# B&R Automation Studio project CControl_Gschneitner (part 8)

#### fbRestzeit.st
```iecst
(* Funktionsbaustein zur Berechnung der Restzeit Lauf/Pause aus 24h Zeitfenstern (BOOL [24]) *)
FUNCTION_BLOCK fbRestzeit

	IF Freigabe THEN

		//Variable setzen, wenn Zeitfenster aktiv
		ZeitfensterAktiv	:= ZeitfensterIn[AktuelleStunde];

		//Zeitfenster ist aktiv -> Restzeit Lauf berechnen *********************************************************
		IF ZeitfensterAktiv THEN

			//Änderung von Struktur Zeitfenster erkennen
			loc_Aenderung := memcmp(ADR(ZeitfensterIn), ADR(MEM_ZeitfensterIn), SIZEOF(ZeitfensterIn));
			IF loc_Aenderung <> 0 OR loc_firstInitLauf THEN
				loc_firstInitLauf := FALSE;
				loc_StundeEndeZeitfTag := 23;
				loc_StundeEndeZeitfFolgetag := 23;
				memcpy(ADR(MEM_ZeitfensterIn), ADR(ZeitfensterIn), SIZEOF(MEM_ZeitfensterIn));
			END_IF

			//Minuten Rest aktueller Tag berechnen
			loc_MinutenRestTag	:= 60 - AktuelleMinute;
			FOR i:= AktuelleStunde + 1 TO loc_StundeEndeZeitfTag DO
				IF ZeitfensterIn[i] = TRUE THEN
					loc_MinutenRestTag	:= loc_MinutenRestTag + 60;
				ELSE
					loc_StundeEndeZeitfTag := i;
				END_IF
			END_FOR

			//Minuten Rest Folgetag berechnen, wenn aktuelles Zeitfenster bis zum Ende des Tages aktiv ist
			loc_MinutenRestFolgetag := 0;
			IF loc_StundeEndeZeitfTag = 23 THEN
				FOR ii:= 0 TO loc_StundeEndeZeitfFolgetag DO
					IF ZeitfensterIn[ii] = TRUE THEN
						loc_MinutenRestFolgetag	:= loc_MinutenRestFolgetag + 60;
					ELSE
						loc_StundeEndeZeitfFolgetag := ii;
					END_IF
				END_FOR
			ELSE
				loc_MinutenRestFolgetag := 0;
				loc_StundeEndeZeitfFolgetag := 23;
			END_IF

			//Gesamtzeit Minuten Tag + Folgetag
			loc_MinutenRestGesamt := loc_MinutenRestTag + loc_MinutenRestFolgetag;

			//Ausgabe Restzeit in Stunden und Minuten
			loc_RestzeitStunden		:= loc_MinutenRestGesamt / 60;
			//Wenn Restzeit Stunden > 24h, Ausgabe Stunden = 255 (keine Anzeige in Visu)
			IF loc_RestzeitStunden <= 24 THEN
				RestzeitStundenOut		:= ABS(loc_RestzeitStunden);
				RestzeitMinutenOut		:= loc_MinutenRestGesamt - (RestzeitStundenOut * 60);
			ELSE
				RestzeitStundenOut		:= 65535;
				RestzeitMinutenOut		:= 65535;
			END_IF

			loc_firstInitPause := TRUE;

		//Zeitfenster nicht aktiv -> Restzeit Pause berechnen *********************************************************
		ELSE

			//Änderung von Struktur Zeitfenster erkennen
			loc_Aenderung := memcmp(ADR(ZeitfensterIn), ADR(MEM_ZeitfensterIn), SIZEOF(ZeitfensterIn));
			IF loc_Aenderung <> 0 OR loc_firstInitPause THEN
				loc_firstInitPause := FALSE;
				loc_StundeEndeZeitfTag := 23;
				loc_StundeEndeZeitfFolgetag := 23;
				memcpy(ADR(MEM_ZeitfensterIn), ADR(ZeitfensterIn), SIZEOF(MEM_ZeitfensterIn));
			END_IF

			//Minuten Rest aktueller Tag berechnen
			loc_MinutenRestTag	:= 60 - AktuelleMinute;
			FOR i:= AktuelleStunde + 1 TO loc_StundeEndeZeitfTag DO
				IF ZeitfensterIn[i] = FALSE THEN
					loc_MinutenRestTag	:= loc_MinutenRestTag + 60;
				ELSE
					loc_StundeEndeZeitfTag := i;
				END_IF
			END_FOR

			//Minuten Rest Folgetag berechnen, wenn aktuelles Zeitfenster bis zum Ende des Tages inaktiv ist
			loc_MinutenRestFolgetag := 0;
			IF loc_StundeEndeZeitfTag = 23 THEN
				FOR ii:= 0 TO loc_StundeEndeZeitfFolgetag DO
					IF ZeitfensterIn[ii] = FALSE THEN
						loc_MinutenRestFolgetag	:= loc_MinutenRestFolgetag + 60;
					ELSE
						loc_StundeEndeZeitfFolgetag := ii;
					END_IF
				END_FOR
			ELSE
				loc_MinutenRestFolgetag := 0;
				loc_StundeEndeZeitfFolgetag := 23;
			END_IF

			//Gesamtzeit Minuten Tag + Folgetag
			loc_MinutenRestGesamt := loc_MinutenRestTag + loc_MinutenRestFolgetag;

			//Ausgabe Restzeit in Stunden und Minuten
			loc_RestzeitStunden		:= loc_MinutenRestGesamt / 60;

			//Wenn Restzeit Stunden > 24h, Ausgabe Stunden = 65535 (keine Anzeige in Visu)
			IF loc_RestzeitStunden <= 24 THEN
				RestzeitStundenOut		:= ABS(loc_RestzeitStunden);
				RestzeitMinutenOut		:= loc_MinutenRestGesamt - (RestzeitStundenOut * 60);
			ELSE
				RestzeitStundenOut		:= 65535;
				RestzeitMinutenOut		:= 65535;
			END_IF

			loc_firstInitLauf := TRUE;

		END_IF

	//Keine Freigabe Baustein
	ELSE

		loc_firstInitLauf	:= TRUE;
		loc_firstInitPause	:= TRUE;
		RestzeitMinutenOut	:= 65535;
		RestzeitStundenOut	:= 65535;

	END_IF

END_FUNCTION_BLOCK
```

### Library Logical/Libraries/IecCheck (IEC)
Depends on: sys_lib, AsBrStr

#### IecCheck.fun - Exported functions and function blocks
```iecst
FUNCTION CheckDivSint : SINT (* Check divisor for SINT division *)
	VAR_INPUT
		divisor : SINT;
	END_VAR
END_FUNCTION

FUNCTION CheckDivUsint : USINT (* Check divisor for USINT division *)
	VAR_INPUT
		divisor : USINT;
	END_VAR
END_FUNCTION

FUNCTION CheckDivInt : INT (* Check divisor for INT division *)
	VAR_INPUT
		divisor : INT;
	END_VAR
END_FUNCTION

FUNCTION CheckDivUint : UINT (* Check divisor for UINT division *)
	VAR_INPUT
		divisor : UINT;
	END_VAR
END_FUNCTION

FUNCTION CheckDivDint : DINT (* Check divisor for DINT division *)
	VAR_INPUT
		divisor : DINT;
	END_VAR
END_FUNCTION

FUNCTION CheckDivUdint : UDINT (* Check divisor for UDINT division *)
	VAR_INPUT
		divisor : UDINT;
	END_VAR
END_FUNCTION

FUNCTION CheckDivReal : REAL (* Check divisor for REAL division *)
	VAR_INPUT
		divisor : REAL;
	END_VAR
END_FUNCTION

FUNCTION CheckDivLReal : LREAL (* Check divisor for LREAL division, not available for SG3 and SGC *)
	VAR_INPUT
		divisor : LREAL;
	END_VAR
END_FUNCTION

FUNCTION CheckBounds : DINT (* Check range for array access *)
	VAR_INPUT
		index : DINT;
		lower : DINT;
		upper : DINT;
	END_VAR
END_FUNCTION

FUNCTION CheckRange : DINT (* Check range for enumeration *)
	VAR_INPUT
		value : DINT;
		lower : DINT;
		upper : DINT;
	END_VAR
END_FUNCTION

FUNCTION CheckSignedSubrange : DINT (* Check range for subrange of signed data types *)
	VAR_INPUT
		value : DINT;
		lower : DINT;
		upper : DINT;
	END_VAR
END_FUNCTION

FUNCTION CheckUnsignedSubrange : UDINT (* Check range for subrange of unsigned data types *)
	VAR_INPUT
		value : UDINT;
		lower : UDINT;
		upper : UDINT;
	END_VAR
END_FUNCTION

FUNCTION CheckReadAccess : UDINT (* Check address when reading dynamic variables *)
	VAR_INPUT
		address : UDINT;
	END_VAR
END_FUNCTION

FUNCTION CheckWriteAccess : UDINT (* Check address when writing dynamic variables *)
	VAR_INPUT
		address : UDINT;
	END_VAR
END_FUNCTION

FUNCTION MakeEntry : UDINT (* Makes an entry (log book entry) in the error log book *)
	VAR
		taskname : STRING[30];
		group : USINT;
		status_name : UINT;
		out_text : STRING[80];
	END_VAR
	VAR_INPUT
		number : UINT;
		index : DINT;
		text : STRING[50];
	END_VAR
END_FUNCTION
```

#### IecCheck.st - Implementation file
```iecst
(* Check divisor for SINT division *)
FUNCTION CheckDivSint
	IF divisor=0 THEN
		CheckDivSint:=1;
		MakeEntry(55555,divisor,'CheckDivSint');
	ELSE
		CheckDivSint:=divisor;
	END_IF
END_FUNCTION

(* Check divisor for USINT division *)
FUNCTION CheckDivUsint
	IF divisor=0 THEN
		CheckDivUsint:=1;
		MakeEntry(55555,divisor,'CheckDivUsint');
	ELSE
		CheckDivUsint:=divisor;
	END_IF
END_FUNCTION

(* Check divisor for INT division *)
FUNCTION CheckDivInt
	IF divisor=0 THEN
		CheckDivInt:=1;
		MakeEntry(55555,divisor,'CheckDivInt');
	ELSE
		CheckDivInt:=divisor;
	END_IF
END_FUNCTION

(* Check divisor for UINT division *)
FUNCTION CheckDivUint
	IF divisor=0 THEN
		CheckDivUint:=1;
		MakeEntry(55555,divisor,'CheckDivUint');
	ELSE
		CheckDivUint:=divisor;
	END_IF
END_FUNCTION

(* Check divisor for DINT division *)
FUNCTION CheckDivDint
	IF divisor=0 THEN
		CheckDivDint:=1;
		MakeEntry(55555,divisor,'CheckDivDint');
	ELSE
		CheckDivDint:=divisor;
	END_IF
END_FUNCTION

(* Check divisor for UDINT division *)
FUNCTION CheckDivUdint
	IF divisor=0 THEN
		CheckDivUdint:=1;
		MakeEntry(55555,divisor,'CheckDivUdint');
	ELSE
		CheckDivUdint:=divisor;
	END_IF
END_FUNCTION

(* Check divisor for REAL division *)
FUNCTION CheckDivReal
	IF divisor=0 THEN
		CheckDivReal:=1;
		MakeEntry(55555,0,'CheckDivReal');
	ELSE
		CheckDivReal:=divisor;
	END_IF
END_FUNCTION

(* Check divisor for LREAL division *)
FUNCTION CheckDivLReal
	IF divisor=0 THEN
		CheckDivLReal:=1;
		MakeEntry(55555,0,'CheckDivLReal');
	ELSE
		CheckDivLReal:=divisor;
	END_IF
END_FUNCTION

(* Check range for array access *)
FUNCTION CheckBounds
	IF index < lower THEN
		CheckBounds := lower;
		MakeEntry(55555,index,'CheckBounds');
	ELSIF index > upper THEN
		CheckBounds := upper;
		MakeEntry(55555,index,'CheckBounds');
	ELSE
		CheckBounds := index;
	END_IF
END_FUNCTION

(* Check range for enumeration *)
FUNCTION CheckRange
	IF value < lower THEN
		CheckRange := lower;
		MakeEntry(55555,value,'CheckRange');
	ELSIF value > upper THEN
		CheckRange := upper;
		MakeEntry(55555,value,'CheckRange');
	ELSE
		CheckRange := value;
	END_IF
END_FUNCTION

(* Check range for subrange of signed data types *)
FUNCTION CheckSignedSubrange
	IF value < lower THEN
		CheckSignedSubrange := lower;
		MakeEntry(55555,value,'CheckSignedSubrange');
	ELSIF value > upper THEN
		CheckSignedSubrange := upper;
		MakeEntry(55555,value,'CheckSignedSubrange');
	ELSE
		CheckSignedSubrange := value;
	END_IF
END_FUNCTION

(* Check range for subrange of unsigned data types *)
FUNCTION CheckUnsignedSubrange
	IF value < lower THEN
		CheckUnsignedSubrange := lower;
		MakeEntry(55555,value,'CheckUnsignedSubrange');
	ELSIF value > upper THEN
		CheckUnsignedSubrange := upper;
		MakeEntry(55555,value,'CheckUnsignedSubrange');
	ELSE
		CheckUnsignedSubrange := value;
	END_IF
END_FUNCTION

(* Check address when reading dynamic variables *)
FUNCTION CheckReadAccess
	IF address=0 THEN
		(* TODO: Insert an appropriate code, see AutomationStudio help for further information *)
		MakeEntry(55555,address,'Read from NULL');
	END_IF

	CheckReadAccess:=0;
END_FUNCTION

(* Check address when writing dynamic variables *)
FUNCTION CheckWriteAccess
	IF address=0 THEN
		(* TODO: Insert an appropriate code, see AutomationStudio help for further information *)
		MakeEntry(55555,address,'Write to NULL');
	END_IF

	CheckWriteAccess:=0;
END_FUNCTION

(* Makes an entry (log book entry) in the error log book *)
FUNCTION MakeEntry
		status_name := ST_name(0,ADR(taskname),ADR(group));

		brsstrcpy(ADR(out_text),ADR(text));
		brsstrcat(ADR(out_text),ADR(' > in task > '));
  		brsstrcat(ADR(out_text),ADR(taskname));
		MakeEntry := ADR(out_text);
		ERRxfatal(number,index,ADR(out_text));
END_FUNCTION
```

### Library Logical/Libraries/CControl (IEC)

#### CControl.fun - Exported functions and function blocks
```iecst
{REDUND_ERROR} {REDUND_UNREPLICABLE} FUNCTION_BLOCK fbCControlWitterung (*Funktionsbaustein zur Generierung der Witterungsverhältnisse über Sättigungsdefizit und Trocknungslaufzeit*) (*$GROUP=User,$CAT=User,$GROUPICON=User.png,$CATICON=User.png*)
	VAR_INPUT
		Freigabe : {REDUND_UNREPLICABLE} BOOL;
		MaterialfeuchteIst : {REDUND_UNREPLICABLE} UDINT;
		MaterialfeuchteStufe : {REDUND_UNREPLICABLE} ARRAY[1..6] OF UDINT;
		FrischluftSaettigungsdefizit : {REDUND_UNREPLICABLE} REAL;
		DachluftSaettigungsdefizit : {REDUND_UNREPLICABLE} REAL;
		TrockenluftSaettigungsdefizit : {REDUND_UNREPLICABLE} REAL;
		AuswahlSensor : {REDUND_UNREPLICABLE} USINT; (*0= Frischluft, 1= Dachluft, 2= Trockenluft*)
		SensorFrischluftVhd : {REDUND_UNREPLICABLE} BOOL;
		SensorDachluftVhd : {REDUND_UNREPLICABLE} BOOL;
		SensorTrockenluftVhd : {REDUND_UNREPLICABLE} BOOL;
		GrenzwertStufeAktuell : {REDUND_UNREPLICABLE} REAL;
		HystereseGrenzwert : {REDUND_UNREPLICABLE} REAL;
		VerzWetterwechsel : {REDUND_UNREPLICABLE} UDINT; (*Verzögerungszeit Wetterwechsel [ms]*)
		SchlechtwetterPulszeitStufe : {REDUND_UNREPLICABLE} ARRAY[1..6] OF UDINT;
		SchlechtwetterPausezeitStufe : {REDUND_UNREPLICABLE} ARRAY[1..6] OF UDINT;
	END_VAR
	VAR_OUTPUT
		StufeAktuell : {REDUND_UNREPLICABLE} USINT;
		WetterIstGut : {REDUND_UNREPLICABLE} BOOL;
		WetterIstSchlecht : {REDUND_UNREPLICABLE} BOOL;
		SchlechtwetterPulszeit : {REDUND_UNREPLICABLE} UDINT;
		SchlechtwetterPausezeit : {REDUND_UNREPLICABLE} UDINT;
	END_VAR
	VAR
		i : {REDUND_UNREPLICABLE} USINT;
		SaettigungsdefizitIst : {REDUND_UNREPLICABLE} REAL;
		loc_WetterIstGut : {REDUND_UNREPLICABLE} BOOL;
		loc_WetterIstSchlecht : {REDUND_UNREPLICABLE} BOOL;
		TON_SchrittWitterung : {REDUND_UNREPLICABLE} TON;
		curStep : {REDUND_UNREPLICABLE} USINT;
		stateEntry : {REDUND_UNREPLICABLE} BOOL;
	END_VAR
END_FUNCTION_BLOCK
```

#### fbCControlWitterung.st
```iecst
(* Funktionsbaustein zur Generierung der Witterungsverhältnisse über Sättigungsdefizit und Trocknungslaufzeit *)
FUNCTION_BLOCK fbCControlWitterung

	IF Freigabe THEN

		//Aktuell gültige Stufe anhand der Trockengutfeuchte ermitteln
		StufeAktuell := 1;
		IF MaterialfeuchteIst <> 0 THEN
			FOR i := 1 TO 5 DO
				IF MaterialfeuchteIst <= MaterialfeuchteStufe[i] THEN
					StufeAktuell := i + 1;
				END_IF
			END_FOR
		END_IF

		//Puls/Pausezeiten für die aktuelle Stufe an Bausteinausgänge übergeben
		SchlechtwetterPulszeit	:= SchlechtwetterPulszeitStufe[StufeAktuell];
		SchlechtwetterPausezeit	:= SchlechtwetterPausezeitStufe[StufeAktuell];

		//Bestimmung gültiger Sensor
		IF (AuswahlSensor = 0) AND SensorFrischluftVhd THEN
			SaettigungsdefizitIst := FrischluftSaettigungsdefizit;
		ELSIF (AuswahlSensor = 1) AND SensorDachluftVhd THEN
			SaettigungsdefizitIst := DachluftSaettigungsdefizit;
		ELSIF (AuswahlSensor = 2) AND SensorTrockenluftVhd THEN
			SaettigungsdefizitIst := TrockenluftSaettigungsdefizit;
		ELSIF SensorFrischluftVhd THEN
			SaettigungsdefizitIst := FrischluftSaettigungsdefizit; //Ausgewählter Sensor nicht vhd. -> Frischluft verwenden
		ELSE
			SaettigungsdefizitIst := 0.0; //Kein Sensor vhd.
		END_IF

		//Witterungsverhältnisse bestimmen
		IF SaettigungsdefizitIst <> 0 THEN

			loc_WetterIstGut		:= FALSE;
			loc_WetterIstSchlecht	:= FALSE;
			IF (SaettigungsdefizitIst >= (GrenzwertStufeAktuell + HystereseGrenzwert)) THEN
				loc_WetterIstGut := TRUE;
			ELSIF (SaettigungsdefizitIst <= (GrenzwertStufeAktuell - HystereseGrenzwert)) THEN
				loc_WetterIstSchlecht := TRUE;
			END_IF

			CASE curStep OF

				//INIT
				0:
					IF stateEntry THEN
						stateEntry := FALSE;
						TON_SchrittWitterung(IN:= FALSE);
					END_IF

					IF loc_WetterIstGut THEN
						curStep := 1;
					ELSE
						curStep := 2;
					END_IF

					//Wetter ist gut
				1:
					IF stateEntry THEN
						stateEntry := FALSE;
						TON_SchrittWitterung(IN:= FALSE);
					END_IF

					WetterIstGut := TRUE;
					WetterIstSchlecht := FALSE;

					TON_SchrittWitterung(IN:= loc_WetterIstSchlecht, PT:= UDINT_TO_TIME(VerzWetterwechsel));

					IF TON_SchrittWitterung.Q THEN
						stateEntry := TRUE;
						curStep := 2;
					END_IF

					//Wetter ist schlecht
				2:

					IF stateEntry THEN
						stateEntry := FALSE;
						TON_SchrittWitterung(IN:= FALSE);
					END_IF

					WetterIstGut := FALSE;
					WetterIstSchlecht := TRUE;

					TON_SchrittWitterung(IN:= loc_WetterIstGut, PT:= UDINT_TO_TIME(VerzWetterwechsel));

					IF TON_SchrittWitterung.Q THEN
						stateEntry := TRUE;
						curStep := 1;
					END_IF

			END_CASE

		ELSE
			loc_WetterIstGut		:= FALSE;
			loc_WetterIstSchlecht	:= FALSE;
			WetterIstGut			:= TRUE;
			WetterIstSchlecht 		:= FALSE;
			TON_SchrittWitterung(IN:= FALSE);
			stateEntry := TRUE;
			curStep := 0;
		END_IF

		//keine Freigabe des Bausteins
	ELSE
		loc_WetterIstGut		:= FALSE;
		loc_WetterIstSchlecht	:= FALSE;
		WetterIstGut			:= FALSE;
		WetterIstSchlecht 		:= FALSE;
		TON_SchrittWitterung(IN:= FALSE);
		stateEntry := TRUE;
		curStep := 0;
		SaettigungsdefizitIst := 0.0;
		SchlechtwetterPulszeit := 0;
		SchlechtwetterPausezeit := 0;
		StufeAktuell := 1;

	END_IF

END_FUNCTION_BLOCK
```

### Package Logical/Util - System, Uhr, Datensicherung

### Program Logical/Util/eUhr (IEC) - Echtzeituhr

#### eUhrCyclic.st - Zyklischer Code
```iecst
PROGRAM _CYCLIC

	//Funktionsbaustein Echtzeituhr
	//=============================

	//Echtzeituhr auslesen
	RTC_gettime(ADR(Echtzeit));

	//Datum und Uhrzeit auslesen
	DTGetTime_0.enable	:= TRUE;
	DTGetTime_0();
	DateTime			:= DTGetTime_0.DT1;

	//Zeit als Word bilden
	Echtzeit.StdMin		:= (Echtzeit.Stunde * 100) + Echtzeit.Minute;

END_PROGRAM
```

#### eUhr.var - Lokale Variablen
```iecst
VAR
	DTGetTime_0 : {REDUND_UNREPLICABLE} DTGetTime;
END_VAR
```

### Program Logical/Util/Nutzung (IEC) - Betriebsstunden, Serviceintervalle

#### Nutzung.st - Zyklischer Code
```iecst
PROGRAM _INIT

	initOk		:= FALSE;
	stateEntry	:= TRUE;

END_PROGRAM

PROGRAM _CYCLIC

	//Nutzungsdaten auswerten
	//=======================

	//Ticks erstellen
	//***************
	fbLascoZdxx_0(IN 	:= Echtzeit.Sekunde);
	sekTick				:= fbLascoZdxx_0.Q;

	fbLascoZdxx_1(IN 	:= Echtzeit.Minute);
	minTick				:= fbLascoZdxx_1.Q;

	fbLascoZdxx_2(IN	:= Echtzeit.Tag);
	tagTick				:= fbLascoZdxx_2.Q;

	fbLascoZdxx_3(IN	:= Echtzeit.Monat);
	monatTick			:= fbLascoZdxx_3.Q;

	fbLascoZdxx_4(IN	:= Echtzeit.Jahr);
	jahrTick			:= fbLascoZdxx_4.Q;

	//======================================================================================================================================================
	//Laufzeit Ölsumpfheizung überwachen
	//======================================================================================================================================================

	IF initOk AND stateEntry THEN
		stateEntry	:= FALSE;

		loc_UhrzeitAktuellUdint	:= DT_TO_UDINT(DTGetTime_0.DT1);
		loc_UhrzeitMEM_Udint	:= DT_TO_UDINT(hmiNutzungsdaten.Allgemein.DatumLetzterBetrieb);
		loc_ZeitStromausfall	:= (loc_UhrzeitAktuellUdint - loc_UhrzeitMEM_Udint) * 1000;

		//Wenn Max. Zeit Stromlos überschritten -> Neustart Mindestlaufzeit Ölsumpfheizung
		IF loc_ZeitStromausfall > Betriebsparameter.Entfeuchter.MaxZeitStromlos THEN
			gMindestlaufzOelsumpfOk	:= FALSE;
			loc_MinLaufzeitOelsumpf	:= Betriebsparameter.Entfeuchter.MindestlaufzeitOelsumpf;
		ELSIF NOT gMindestlaufzOelsumpfOk THEN
			//Doppelte Zeit Stromausfall + Restlaufzeit kleiner Mindestlaufzeit -> Restzeit + Zeit Stromausfall *2
			IF (Betriebsparameter.Entfeuchter.RestzeitLaufzOelsumpf + (loc_ZeitStromausfall * 2)) <
				Betriebsparameter.Entfeuchter.MindestlaufzeitOelsumpf THEN
				loc_MinLaufzeitOelsumpf	:= Betriebsparameter.Entfeuchter.RestzeitLaufzOelsumpf + (loc_ZeitStromausfall * 2);
			ELSE
				loc_MinLaufzeitOelsumpf	:= Betriebsparameter.Entfeuchter.MindestlaufzeitOelsumpf;
			END_IF
		ELSE
			loc_MinLaufzeitOelsumpf	:= 0;
		END_IF
	END_IF

	//Mindestlaufzeit Ölsumpfheizung starten, wenn Ölsumpfheizung aktiv
	TON_MinLaufzeitOelsumpfh(IN:= doOelsumpfheizungEinModul1 AND initOk AND NOT stateEntry, PT:= loc_MinLaufzeitOelsumpf);
	IF TON_MinLaufzeitOelsumpfh.Q THEN
		gMindestlaufzOelsumpfOk	:= TRUE;
	END_IF

	//Aktuelle Uhrzeit und Restlaufzeit minütlich speichern
	DTGetTime_0(enable := TRUE);
	IF minTick AND initOk AND NOT stateEntry THEN
		hmiNutzungsdaten.Allgemein.DatumLetzterBetrieb			:= DTGetTime_0.DT1;
		hmiParameter.Entfeuchter.RestzeitLaufzOelsumpf		:= loc_MinLaufzeitOelsumpf - TIME_TO_UDINT(TON_MinLaufzeitOelsumpfh.ET);
	END_IF

	//======================================================================================================================================================
	//Betriebsstunden (nicht rückstellbar)
	//======================================================================================================================================================

	//Ventilator 1
	//************
	fbMinutenVentilator1Ges.Aktiv		:= diVentilator1InBetrieb AND doVentilator1Ein;
	fbMinutenVentilator1Ges.sekTick		:= sekTick;
	fbMinutenVentilator1Ges.Minuten		:= ADR(hmiNutzungsdaten.BstGes.Ventilator1Min);
	fbMinutenVentilator1Ges();

	fbStundenVentilator1Ges.Minuten		:= ADR(hmiNutzungsdaten.BstGes.Ventilator1Min);
	fbStundenVentilator1Ges.Stunden		:= ADR(hmiNutzungsdaten.BstGes.Ventilator1Std);
	fbStundenVentilator1Ges();

	//Ventilator 2
	//************
	fbMinutenVentilator2Ges.Aktiv		:= diVentilator2InBetrieb AND doVentilator2Ein;
	fbMinutenVentilator2Ges.sekTick		:= sekTick;
	fbMinutenVentilator2Ges.Minuten		:= ADR(hmiNutzungsdaten.BstGes.Ventilator2Min);
	fbMinutenVentilator2Ges();

	fbStundenVentilator2Ges.Minuten		:= ADR(hmiNutzungsdaten.BstGes.Ventilator2Min);
	fbStundenVentilator2Ges.Stunden		:= ADR(hmiNutzungsdaten.BstGes.Ventilator2Std);
	fbStundenVentilator2Ges();

	//Ölsumpfheizung
	//**************
	fbMinutenOelsumpfhGes.Aktiv			:= doOelsumpfheizungEinModul1;
	fbMinutenOelsumpfhGes.sekTick		:= sekTick;
	fbMinutenOelsumpfhGes.Minuten		:= ADR(hmiNutzungsdaten.BstGes.OelsumpfheizungMin);
	fbMinutenOelsumpfhGes();

	fbStundenOelsumpfhGes.Minuten		:= ADR(hmiNutzungsdaten.BstGes.OelsumpfheizungMin);
	fbStundenOelsumpfhGes.Stunden		:= ADR(hmiNutzungsdaten.BstGes.OelsumpfheizungStd);
	fbStundenOelsumpfhGes();

	//Kompressor 1
	//************
	fbMinutenKompressor1Ges.Aktiv		:= doKompressorEinModul1 OR doEntfFremdFreigabe; //ab V2.0.0
	fbMinutenKompressor1Ges.sekTick		:= sekTick;
	fbMinutenKompressor1Ges.Minuten		:= ADR(hmiNutzungsdaten.BstGes.Kompressor1Min);
	fbMinutenKompressor1Ges();

	fbStundenKompressor1Ges.Minuten		:= ADR(hmiNutzungsdaten.BstGes.Kompressor1Min);
	fbStundenKompressor1Ges.Stunden		:= ADR(hmiNutzungsdaten.BstGes.Kompressor1Std);
	fbStundenKompressor1Ges();

	//Kompressor 2
	//************
	fbMinutenKompressor2Ges.Aktiv		:= doKompressorEinModul2;
	fbMinutenKompressor2Ges.sekTick		:= sekTick;
	fbMinutenKompressor2Ges.Minuten		:= ADR(hmiNutzungsdaten.BstGes.Kompressor2Min);
	fbMinutenKompressor2Ges();

	fbStundenKompressor2Ges.Minuten		:= ADR(hmiNutzungsdaten.BstGes.Kompressor2Min);
	fbStundenKompressor2Ges.Stunden		:= ADR(hmiNutzungsdaten.BstGes.Kompressor2Std);
	fbStundenKompressor2Ges();

	//Warmluftofen
	//************
	fbMinutenWarmluftofenGes.Aktiv		:= Aktoren.Warmluftofen.WarmluftofenAktiv;
	fbMinutenWarmluftofenGes.sekTick	:= sekTick;
	fbMinutenWarmluftofenGes.Minuten	:= ADR(hmiNutzungsdaten.BstGes.WarmluftofenMin);
	fbMinutenWarmluftofenGes();

	fbStundenWarmluftofenGes.Minuten	:= ADR(hmiNutzungsdaten.BstGes.WarmluftofenMin);
	fbStundenWarmluftofenGes.Stunden	:= ADR(hmiNutzungsdaten.BstGes.WarmluftofenStd);
	fbStundenWarmluftofenGes();

	//Heizregister
	//************
	fbMinutenHeizregisterGes.Aktiv		:= doHeizregisterEin;
	fbMinutenHeizregisterGes.sekTick	:= sekTick;
	fbMinutenHeizregisterGes.Minuten	:= ADR(hmiNutzungsdaten.BstGes.HeizregisterMin);
	fbMinutenHeizregisterGes();

	fbStundenHeizregisterGes.Minuten	:= ADR(hmiNutzungsdaten.BstGes.HeizregisterMin);
	fbStundenHeizregisterGes.Stunden	:= ADR(hmiNutzungsdaten.BstGes.HeizregisterStd);
	fbStundenHeizregisterGes();

	//Scheitholzofen
	//**************
	fbMinutenScheitholzofenGes.Aktiv	:= Aktoren.Scheitholzofen.ScheitholzofenAktiv;
	fbMinutenScheitholzofenGes.sekTick	:= sekTick;
	fbMinutenScheitholzofenGes.Minuten	:= ADR(hmiNutzungsdaten.BstGes.ScheitholzofenMin);
	fbMinutenScheitholzofenGes();

	fbStundenScheitholzofenGes.Minuten	:= ADR(hmiNutzungsdaten.BstGes.ScheitholzofenMin);
	fbStundenScheitholzofenGes.Stunden	:= ADR(hmiNutzungsdaten.BstGes.ScheitholzofenStd);
	fbStundenScheitholzofenGes();

	//Abtauung Modul 1
	//****************
	fbMinutenAbtauung1Ges.Aktiv			:= Aktoren.KompressorModul1.AbtauungAktiv;
	fbMinutenAbtauung1Ges.sekTick		:= sekTick;
	fbMinutenAbtauung1Ges.Minuten		:= ADR(hmiNutzungsdaten.BstGes.Abtauung1Min);
	fbMinutenAbtauung1Ges();

	fbStundenAbtauung1Ges.Minuten		:= ADR(hmiNutzungsdaten.BstGes.Abtauung1Min);
	fbStundenAbtauung1Ges.Stunden		:= ADR(hmiNutzungsdaten.BstGes.Abtauung1Std);
	fbStundenAbtauung1Ges();

	//Abtauung Modul 2
	//****************
	fbMinutenAbtauung2Ges.Aktiv			:= Aktoren.KompressorModul2.AbtauungAktiv;
	fbMinutenAbtauung2Ges.sekTick		:= sekTick;
	fbMinutenAbtauung2Ges.Minuten		:= ADR(hmiNutzungsdaten.BstGes.Abtauung2Min);
	fbMinutenAbtauung2Ges();

	fbStundenAbtauung2Ges.Minuten		:= ADR(hmiNutzungsdaten.BstGes.Abtauung2Min);
	fbStundenAbtauung2Ges.Stunden		:= ADR(hmiNutzungsdaten.BstGes.Abtauung2Std);
	fbStundenAbtauung2Ges();

	//Abluftventilator
	//****************
	fbMinutenAbluftventGes.Aktiv		:= Betriebsparameter.Ausstattung.Abluftventilator AND diAbluftventInBetrieb;
	fbMinutenAbluftventGes.sekTick		:= sekTick;
	fbMinutenAbluftventGes.Minuten		:= ADR(hmiNutzungsdaten.BstGes.AbluftventMin);
	fbMinutenAbluftventGes();

	fbStundenAbluftventGes.Minuten		:= ADR(hmiNutzungsdaten.BstGes.AbluftventMin);
	fbStundenAbluftventGes.Stunden		:= ADR(hmiNutzungsdaten.BstGes.AbluftventStd);
	fbStundenAbluftventGes();

	//Frischluftbetrieb
	//*****************
	fbMinutenFrischluftbetrGes.Aktiv		:= gStatusAnlage.FrischluftbetriebAktiv AND (gAktModus = BETRIEB);
	fbMinutenFrischluftbetrGes.sekTick		:= sekTick;
	fbMinutenFrischluftbetrGes.Minuten		:= ADR(hmiNutzungsdaten.BstGes.FrischluftbetrMin);
	fbMinutenFrischluftbetrGes();

	fbStundenFrischluftbetrGes.Minuten		:= ADR(hmiNutzungsdaten.BstGes.FrischluftbetrMin);
	fbStundenFrischluftbetrGes.Stunden		:= ADR(hmiNutzungsdaten.BstGes.FrischluftbetrStd);
	fbStundenFrischluftbetrGes();

	//Umluftbetrieb
	//*************
	fbMinutenUmluftbetrGes.Aktiv		:= gStatusAnlage.UmluftbetriebAktiv AND (gAktModus = BETRIEB);
	fbMinutenUmluftbetrGes.sekTick		:= sekTick;
	fbMinutenUmluftbetrGes.Minuten		:= ADR(hmiNutzungsdaten.BstGes.UmluftbetrMin);
	fbMinutenUmluftbetrGes();

	fbStundenUmluftbetrGes.Minuten		:= ADR(hmiNutzungsdaten.BstGes.UmluftbetrMin);
	fbStundenUmluftbetrGes.Stunden		:= ADR(hmiNutzungsdaten.BstGes.UmluftbetrStd);
	fbStundenUmluftbetrGes();

	//Box 1
	//*****
	fbMinutenBox1Ges.Aktiv		:= Boxen.Box1Out.BoxBereit;
	fbMinutenBox1Ges.sekTick	:= sekTick;
	fbMinutenBox1Ges.Minuten	:= ADR(hmiNutzungsdaten.BstGes.Box1Min);
	fbMinutenBox1Ges();

	fbStundenBox1Ges.Minuten	:= ADR(hmiNutzungsdaten.BstGes.Box1Min);
	fbStundenBox1Ges.Stunden	:= ADR(hmiNutzungsdaten.BstGes.Box1Std);
	fbStundenBox1Ges();

	//Box 2
	//*****
	fbMinutenBox2Ges.Aktiv		:= Boxen.Box2Out.BoxBereit;
	fbMinutenBox2Ges.sekTick	:= sekTick;
	fbMinutenBox2Ges.Minuten	:= ADR(hmiNutzungsdaten.BstGes.Box2Min);
	fbMinutenBox2Ges();

	fbStundenBox2Ges.Minuten	:= ADR(hmiNutzungsdaten.BstGes.Box2Min);
	fbStundenBox2Ges.Stunden	:= ADR(hmiNutzungsdaten.BstGes.Box2Std);
	fbStundenBox2Ges();

	//Box 3
	//*****
	fbMinutenBox3Ges.Aktiv		:= Boxen.Box3Out.BoxBereit;
	fbMinutenBox3Ges.sekTick	:= sekTick;
	fbMinutenBox3Ges.Minuten	:= ADR(hmiNutzungsdaten.BstGes.Box3Min);
	fbMinutenBox3Ges();

	fbStundenBox3Ges.Minuten	:= ADR(hmiNutzungsdaten.BstGes.Box3Min);
	fbStundenBox3Ges.Stunden	:= ADR(hmiNutzungsdaten.BstGes.Box3Std);
	fbStundenBox3Ges();

	//Box 4
	//*****
	fbMinutenBox4Ges.Aktiv		:= Boxen.Box4Out.BoxBereit;
	fbMinutenBox4Ges.sekTick	:= sekTick;
	fbMinutenBox4Ges.Minuten	:= ADR(hmiNutzungsdaten.BstGes.Box4Min);
	fbMinutenBox4Ges();

	fbStundenBox4Ges.Minuten	:= ADR(hmiNutzungsdaten.BstGes.Box4Min);
	fbStundenBox4Ges.Stunden	:= ADR(hmiNutzungsdaten.BstGes.Box4Std);
	fbStundenBox4Ges();

	//Box 5
	//*****
	fbMinutenBox5Ges.Aktiv		:= Boxen.Box5Out.BoxBereit;
	fbMinutenBox5Ges.sekTick	:= sekTick;
	fbMinutenBox5Ges.Minuten	:= ADR(hmiNutzungsdaten.BstGes.Box5Min);
	fbMinutenBox5Ges();

	fbStundenBox5Ges.Minuten	:= ADR(hmiNutzungsdaten.BstGes.Box5Min);
	fbStundenBox5Ges.Stunden	:= ADR(hmiNutzungsdaten.BstGes.Box5Std);
	fbStundenBox5Ges();

	//Box 6
	//*****
	fbMinutenBox6Ges.Aktiv		:= Boxen.Box6Out.BoxBereit;
	fbMinutenBox6Ges.sekTick	:= sekTick;
	fbMinutenBox6Ges.Minuten	:= ADR(hmiNutzungsdaten.BstGes.Box6Min);
	fbMinutenBox6Ges();

	fbStundenBox6Ges.Minuten	:= ADR(hmiNutzungsdaten.BstGes.Box6Min);
	fbStundenBox6Ges.Stunden	:= ADR(hmiNutzungsdaten.BstGes.Box6Std);
	fbStundenBox6Ges();

	//======================================================================================================================================================
	//Betriebsstunden (rückstellbar)
	//======================================================================================================================================================

	//Ventilator 1
	//************
	fbMinutenVentilator1.Aktiv		:= diVentilator1InBetrieb AND doVentilator1Ein;
	fbMinutenVentilator1.sekTick	:= sekTick;
	fbMinutenVentilator1.Minuten	:= ADR(hmiNutzungsdaten.Bst.Ventilator1Min);
	fbMinutenVentilator1();

	fbStundenVentilator1.Minuten	:= ADR(hmiNutzungsdaten.Bst.Ventilator1Min);
	fbStundenVentilator1.Stunden	:= ADR(hmiNutzungsdaten.Bst.Ventilator1Std);
	fbStundenVentilator1();

	//Ventilator 2
	//************
	fbMinutenVentilator2.Aktiv		:= diVentilator2InBetrieb AND doVentilator2Ein;
	fbMinutenVentilator2.sekTick	:= sekTick;
	fbMinutenVentilator2.Minuten	:= ADR(hmiNutzungsdaten.Bst.Ventilator2Min);
	fbMinutenVentilator2();

	fbStundenVentilator2.Minuten	:= ADR(hmiNutzungsdaten.Bst.Ventilator2Min);
	fbStundenVentilator2.Stunden	:= ADR(hmiNutzungsdaten.Bst.Ventilator2Std);
	fbStundenVentilator2();

	//Ölsumpfheizung
	//**************
	fbMinutenOelsumpfh.Aktiv		:= doOelsumpfheizungEinModul1;
	fbMinutenOelsumpfh.sekTick		:= sekTick;
	fbMinutenOelsumpfh.Minuten		:= ADR(hmiNutzungsdaten.Bst.OelsumpfheizungMin);
	fbMinutenOelsumpfh();

	fbStundenOelsumpfh.Minuten		:= ADR(hmiNutzungsdaten.Bst.OelsumpfheizungMin);
	fbStundenOelsumpfh.Stunden		:= ADR(hmiNutzungsdaten.Bst.OelsumpfheizungStd);
	fbStundenOelsumpfh();

	//Kompressor 1
	//************
	fbMinutenKompressor1.Aktiv			:= doKompressorEinModul1 OR doEntfFremdFreigabe; //ab V2.0.0
	fbMinutenKompressor1.sekTick		:= sekTick;
	fbMinutenKompressor1.Minuten		:= ADR(hmiNutzungsdaten.Bst.Kompressor1Min);
	fbMinutenKompressor1();

	fbStundenKompressor1.Minuten		:= ADR(hmiNutzungsdaten.Bst.Kompressor1Min);
	fbStundenKompressor1.Stunden		:= ADR(hmiNutzungsdaten.Bst.Kompressor1Std);
	fbStundenKompressor1();

	//Kompressor 2
	//************
	fbMinutenKompressor2.Aktiv			:= doKompressorEinModul2;
	fbMinutenKompressor2.sekTick		:= sekTick;
	fbMinutenKompressor2.Minuten		:= ADR(hmiNutzungsdaten.Bst.Kompressor2Min);
	fbMinutenKompressor2();

	fbStundenKompressor2.Minuten		:= ADR(hmiNutzungsdaten.Bst.Kompressor2Min);
	fbStundenKompressor2.Stunden		:= ADR(hmiNutzungsdaten.Bst.Kompressor2Std);
	fbStundenKompressor2();

	//Warmluftofen
	//************
	fbMinutenWarmluftofen.Aktiv		:= Aktoren.Warmluftofen.WarmluftofenAktiv;
	fbMinutenWarmluftofen.sekTick	:= sekTick;
	fbMinutenWarmluftofen.Minuten	:= ADR(hmiNutzungsdaten.Bst.WarmluftofenMin);
	fbMinutenWarmluftofen();

	fbStundenWarmluftofen.Minuten	:= ADR(hmiNutzungsdaten.Bst.WarmluftofenMin);
	fbStundenWarmluftofen.Stunden	:= ADR(hmiNutzungsdaten.Bst.WarmluftofenStd);
	fbStundenWarmluftofen();

	//Heizregister
	//************
	fbMinutenHeizregister.Aktiv		:= doHeizregisterEin;
	fbMinutenHeizregister.sekTick	:= sekTick;
	fbMinutenHeizregister.Minuten	:= ADR(hmiNutzungsdaten.Bst.HeizregisterMin);
	fbMinutenHeizregister();

	fbStundenHeizregister.Minuten	:= ADR(hmiNutzungsdaten.Bst.HeizregisterMin);
	fbStundenHeizregister.Stunden	:= ADR(hmiNutzungsdaten.Bst.HeizregisterStd);
	fbStundenHeizregister();

	//Scheitholzofen
	//**************
	fbMinutenScheitholzofen.Aktiv	:= Aktoren.Scheitholzofen.ScheitholzofenAktiv;
	fbMinutenScheitholzofen.sekTick	:= sekTick;
	fbMinutenScheitholzofen.Minuten	:= ADR(hmiNutzungsdaten.Bst.ScheitholzofenMin);
	fbMinutenScheitholzofen();

	fbStundenScheitholzofen.Minuten	:= ADR(hmiNutzungsdaten.Bst.ScheitholzofenMin);
	fbStundenScheitholzofen.Stunden	:= ADR(hmiNutzungsdaten.Bst.ScheitholzofenStd);
	fbStundenScheitholzofen();

	//Abtauung Modul 1
	//****************
	fbMinutenAbtauung1.Aktiv		:= Aktoren.KompressorModul1.AbtauungAktiv;
	fbMinutenAbtauung1.sekTick		:= sekTick;
	fbMinutenAbtauung1.Minuten		:= ADR(hmiNutzungsdaten.Bst.Abtauung1Min);
	fbMinutenAbtauung1();

	fbStundenAbtauung1.Minuten		:= ADR(hmiNutzungsdaten.Bst.Abtauung1Min);
	fbStundenAbtauung1.Stunden		:= ADR(hmiNutzungsdaten.Bst.Abtauung1Std);
	fbStundenAbtauung1();

	//Abtauung Modul 2
	//****************
	fbMinutenAbtauung2.Aktiv		:= Aktoren.KompressorModul2.AbtauungAktiv;
	fbMinutenAbtauung2.sekTick		:= sekTick;
	fbMinutenAbtauung2.Minuten		:= ADR(hmiNutzungsdaten.Bst.Abtauung2Min);
	fbMinutenAbtauung2();

	fbStundenAbtauung2.Minuten		:= ADR(hmiNutzungsdaten.Bst.Abtauung2Min);
	fbStundenAbtauung2.Stunden		:= ADR(hmiNutzungsdaten.Bst.Abtauung2Std);
	fbStundenAbtauung2();

	//Abluftventilator
	//****************
	fbMinutenAbluftvent.Aktiv		:= Betriebsparameter.Ausstattung.Abluftventilator AND diAbluftventInBetrieb;
	fbMinutenAbluftvent.sekTick		:= sekTick;
	fbMinutenAbluftvent.Minuten		:= ADR(hmiNutzungsdaten.Bst.AbluftventMin);
	fbMinutenAbluftvent();

	fbStundenAbluftvent.Minuten		:= ADR(hmiNutzungsdaten.Bst.AbluftventMin);
	fbStundenAbluftvent.Stunden		:= ADR(hmiNutzungsdaten.Bst.AbluftventStd);
	fbStundenAbluftvent();

	//Frischluftbetrieb
	//*****************
	fbMinutenFrischluftbetr.Aktiv		:= gStatusAnlage.FrischluftbetriebAktiv AND (gAktModus = BETRIEB);
	fbMinutenFrischluftbetr.sekTick		:= sekTick;
	fbMinutenFrischluftbetr.Minuten		:= ADR(hmiNutzungsdaten.Bst.FrischluftbetrMin);
	fbMinutenFrischluftbetr();

	fbStundenFrischluftbetr.Minuten		:= ADR(hmiNutzungsdaten.Bst.FrischluftbetrMin);
	fbStundenFrischluftbetr.Stunden		:= ADR(hmiNutzungsdaten.Bst.FrischluftbetrStd);
	fbStundenFrischluftbetr();

	//Umluftbetrieb
	//*************
	fbMinutenUmluftbetr.Aktiv		:= gStatusAnlage.UmluftbetriebAktiv AND (gAktModus = BETRIEB);
	fbMinutenUmluftbetr.sekTick		:= sekTick;
	fbMinutenUmluftbetr.Minuten		:= ADR(hmiNutzungsdaten.Bst.UmluftbetrMin);
	fbMinutenUmluftbetr();

	fbStundenUmluftbetr.Minuten		:= ADR(hmiNutzungsdaten.Bst.UmluftbetrMin);
	fbStundenUmluftbetr.Stunden		:= ADR(hmiNutzungsdaten.Bst.UmluftbetrStd);
	fbStundenUmluftbetr();

	//======================================================================================================================================================
	//Stundenaufzeichnung für Trocknungsbilanzen (Gesamtstunden, Ventilatorbetrieb, Betrieb mit Luftaufbereitung)
	//======================================================================================================================================================

	//Box 1
	//*******************************************************************************************************************************

	//Gesamt
	fbMinutenBox1.Aktiv		:= Boxen.Box1Out.BoxBereit;
	fbMinutenBox1.sekTick	:= sekTick;
	fbMinutenBox1.Minuten	:= ADR(hmiNutzungsdaten.Bst.Box1Min);
	fbMinutenBox1();

	fbStundenBox1.Minuten	:= ADR(hmiNutzungsdaten.Bst.Box1Min);
	fbStundenBox1.Stunden	:= ADR(hmiNutzungsdaten.Bst.Box1Std);
	fbStundenBox1();

	//Ventilatorbetrieb
	fbMinutenVentBox1.Aktiv := Boxen.Box1Out.BoxBereit AND ((diVentilator1InBetrieb AND Betriebsparameter.Boxen[1].Ventilator1) OR
	(diVentilator2InBetrieb AND Betriebsparameter.Boxen[1].Ventilator2));
	fbMinutenVentBox1.sekTick := sekTick;
	fbMinutenVentBox1.Minuten := ADR(hmiNutzungsdaten.Trocknungsbilanz.VentMinutenBox1);
	fbMinutenVentBox1();

	fbStundenVentBox1.Minuten := ADR(hmiNutzungsdaten.Trocknungsbilanz.VentMinutenBox1);
	fbStundenVentBox1.Stunden := ADR(hmiNutzungsdaten.Trocknungsbilanz.VentStundenBox1);
	fbStundenVentBox1();

	//Betrieb mit Luftaufbereitung
	fbMinutenLuftaufbBox1.Aktiv := Boxen.Box1Out.BoxBereit AND (((diBetriebsmldgKompressorModul1 OR diEntfeuchterFremdInBetrieb) AND Betriebsparameter.Boxen[1].Luftentfeuchter) OR
	(diScheitholzofenInBetrieb AND Betriebsparameter.Boxen[1].Scheitholzofen) OR (doHeizregisterEin AND Betriebsparameter.Boxen[1].Heizregister) OR
	(Aktoren.Warmluftofen.WarmluftofenAktiv AND Betriebsparameter.Boxen[1].Warmluftofen));
	fbMinutenLuftaufbBox1.sekTick := sekTick;
	fbMinutenLuftaufbBox1.Minuten := ADR(hmiNutzungsdaten.Trocknungsbilanz.LuftaufbMinutenBox1);
	fbMinutenLuftaufbBox1();

	fbStundenLuftaufbBox1.Minuten := ADR(hmiNutzungsdaten.Trocknungsbilanz.LuftaufbMinutenBox1);
	fbStundenLuftaufbBox1.Stunden := ADR(hmiNutzungsdaten.Trocknungsbilanz.LuftaufbStundenBox1);
	fbStundenLuftaufbBox1();

	//Box 2
	//*******************************************************************************************************************************

	//Gesamt
	fbMinutenBox2.Aktiv		:= Boxen.Box2Out.BoxBereit;
	fbMinutenBox2.sekTick	:= sekTick;
	fbMinutenBox2.Minuten	:= ADR(hmiNutzungsdaten.Bst.Box2Min);
	fbMinutenBox2();

	fbStundenBox2.Minuten	:= ADR(hmiNutzungsdaten.Bst.Box2Min);
	fbStundenBox2.Stunden	:= ADR(hmiNutzungsdaten.Bst.Box2Std);
	fbStundenBox2();

	//Ventilatorbetrieb
	fbMinutenVentBox2.Aktiv := Boxen.Box2Out.BoxBereit AND ((diVentilator1InBetrieb AND Betriebsparameter.Boxen[2].Ventilator1) OR
	(diVentilator2InBetrieb AND Betriebsparameter.Boxen[2].Ventilator2));
	fbMinutenVentBox2.sekTick := sekTick;
	fbMinutenVentBox2.Minuten := ADR(hmiNutzungsdaten.Trocknungsbilanz.VentMinutenBox2);
	fbMinutenVentBox2();

	fbStundenVentBox2.Minuten := ADR(hmiNutzungsdaten.Trocknungsbilanz.VentMinutenBox2);
	fbStundenVentBox2.Stunden := ADR(hmiNutzungsdaten.Trocknungsbilanz.VentStundenBox2);
	fbStundenVentBox2();

	//Betrieb mit Luftaufbereitung
	fbMinutenLuftaufbBox2.Aktiv := Boxen.Box2Out.BoxBereit AND (((diBetriebsmldgKompressorModul1 OR diEntfeuchterFremdInBetrieb)  AND Betriebsparameter.Boxen[2].Luftentfeuchter) OR
	(diScheitholzofenInBetrieb AND Betriebsparameter.Boxen[2].Scheitholzofen) OR (doHeizregisterEin AND Betriebsparameter.Boxen[2].Heizregister) OR
	(Aktoren.Warmluftofen.WarmluftofenAktiv AND Betriebsparameter.Boxen[2].Warmluftofen)) ;
	fbMinutenLuftaufbBox2.sekTick := sekTick;
	fbMinutenLuftaufbBox2.Minuten := ADR(hmiNutzungsdaten.Trocknungsbilanz.LuftaufbMinutenBox2);
	fbMinutenLuftaufbBox2();

	fbStundenLuftaufbBox2.Minuten := ADR(hmiNutzungsdaten.Trocknungsbilanz.LuftaufbMinutenBox2);
	fbStundenLuftaufbBox2.Stunden := ADR(hmiNutzungsdaten.Trocknungsbilanz.LuftaufbStundenBox2);
	fbStundenLuftaufbBox2();

	//Box 3
	//*******************************************************************************************************************************

	//Gesamt
	fbMinutenBox3.Aktiv		:= Boxen.Box3Out.BoxBereit;
	fbMinutenBox3.sekTick	:= sekTick;
	fbMinutenBox3.Minuten	:= ADR(hmiNutzungsdaten.Bst.Box3Min);
	fbMinutenBox3();

	fbStundenBox3.Minuten	:= ADR(hmiNutzungsdaten.Bst.Box3Min);
	fbStundenBox3.Stunden	:= ADR(hmiNutzungsdaten.Bst.Box3Std);
	fbStundenBox3();

	//Ventilatorbetrieb
	fbMinutenVentBox3.Aktiv := Boxen.Box3Out.BoxBereit AND ((diVentilator1InBetrieb AND Betriebsparameter.Boxen[3].Ventilator1) OR
	(diVentilator2InBetrieb AND Betriebsparameter.Boxen[3].Ventilator2));
	fbMinutenVentBox3.sekTick := sekTick;
	fbMinutenVentBox3.Minuten := ADR(hmiNutzungsdaten.Trocknungsbilanz.VentMinutenBox3);
	fbMinutenVentBox3();

	fbStundenVentBox3.Minuten := ADR(hmiNutzungsdaten.Trocknungsbilanz.VentMinutenBox3);
	fbStundenVentBox3.Stunden := ADR(hmiNutzungsdaten.Trocknungsbilanz.VentStundenBox3);
	fbStundenVentBox3();

	//Betrieb mit Luftaufbereitung
	fbMinutenLuftaufbBox3.Aktiv := Boxen.Box3Out.BoxBereit AND (((diBetriebsmldgKompressorModul1 OR diEntfeuchterFremdInBetrieb)  AND Betriebsparameter.Boxen[3].Luftentfeuchter) OR
	(diScheitholzofenInBetrieb AND Betriebsparameter.Boxen[3].Scheitholzofen) OR (doHeizregisterEin AND Betriebsparameter.Boxen[3].Heizregister) OR
	(Aktoren.Warmluftofen.WarmluftofenAktiv AND Betriebsparameter.Boxen[3].Warmluftofen)) ;
	fbMinutenLuftaufbBox3.sekTick := sekTick;
	fbMinutenLuftaufbBox3.Minuten := ADR(hmiNutzungsdaten.Trocknungsbilanz.LuftaufbMinutenBox3);
	fbMinutenLuftaufbBox3();

	fbStundenLuftaufbBox3.Minuten := ADR(hmiNutzungsdaten.Trocknungsbilanz.LuftaufbMinutenBox3);
	fbStundenLuftaufbBox3.Stunden := ADR(hmiNutzungsdaten.Trocknungsbilanz.LuftaufbStundenBox3);
	fbStundenLuftaufbBox3();

	//Box 4
	//*******************************************************************************************************************************

	//Gesamt
	fbMinutenBox4.Aktiv		:= Boxen.Box4Out.BoxBereit;
	fbMinutenBox4.sekTick	:= sekTick;
	fbMinutenBox4.Minuten	:= ADR(hmiNutzungsdaten.Bst.Box4Min);
	fbMinutenBox4();

	fbStundenBox4.Minuten	:= ADR(hmiNutzungsdaten.Bst.Box4Min);
	fbStundenBox4.Stunden	:= ADR(hmiNutzungsdaten.Bst.Box4Std);
	fbStundenBox4();

	//Ventilatorbetrieb
	fbMinutenVentBox4.Aktiv := Boxen.Box4Out.BoxBereit AND ((diVentilator1InBetrieb AND Betriebsparameter.Boxen[4].Ventilator1) OR
	(diVentilator2InBetrieb AND Betriebsparameter.Boxen[4].Ventilator2));
	fbMinutenVentBox4.sekTick := sekTick;
	fbMinutenVentBox4.Minuten := ADR(hmiNutzungsdaten.Trocknungsbilanz.VentMinutenBox4);
	fbMinutenVentBox4();

	fbStundenVentBox4.Minuten := ADR(hmiNutzungsdaten.Trocknungsbilanz.VentMinutenBox4);
	fbStundenVentBox4.Stunden := ADR(hmiNutzungsdaten.Trocknungsbilanz.VentStundenBox4);
	fbStundenVentBox4();

	//Betrieb mit Luftaufbereitung
	fbMinutenLuftaufbBox4.Aktiv := Boxen.Box4Out.BoxBereit AND (((diBetriebsmldgKompressorModul1 OR diEntfeuchterFremdInBetrieb)  AND Betriebsparameter.Boxen[4].Luftentfeuchter) OR
	(diScheitholzofenInBetrieb AND Betriebsparameter.Boxen[4].Scheitholzofen) OR (doHeizregisterEin AND Betriebsparameter.Boxen[4].Heizregister) OR
	(Aktoren.Warmluftofen.WarmluftofenAktiv AND Betriebsparameter.Boxen[4].Warmluftofen)) ;
	fbMinutenLuftaufbBox4.sekTick := sekTick;
	fbMinutenLuftaufbBox4.Minuten := ADR(hmiNutzungsdaten.Trocknungsbilanz.LuftaufbMinutenBox4);
	fbMinutenLuftaufbBox4();

	fbStundenLuftaufbBox4.Minuten := ADR(hmiNutzungsdaten.Trocknungsbilanz.LuftaufbMinutenBox4);
	fbStundenLuftaufbBox4.Stunden := ADR(hmiNutzungsdaten.Trocknungsbilanz.LuftaufbStundenBox4);
	fbStundenLuftaufbBox4();

	//Box 5
	//*******************************************************************************************************************************

	//Gesamt
	fbMinutenBox5.Aktiv		:= Boxen.Box5Out.BoxBereit;
	fbMinutenBox5.sekTick	:= sekTick;
	fbMinutenBox5.Minuten	:= ADR(hmiNutzungsdaten.Bst.Box5Min);
	fbMinutenBox5();

	fbStundenBox5.Minuten	:= ADR(hmiNutzungsdaten.Bst.Box5Min);
	fbStundenBox5.Stunden	:= ADR(hmiNutzungsdaten.Bst.Box5Std);
	fbStundenBox5();

	//Ventilatorbetrieb
	fbMinutenVentBox5.Aktiv := Boxen.Box5Out.BoxBereit AND ((diVentilator1InBetrieb AND Betriebsparameter.Boxen[5].Ventilator1) OR
	(diVentilator2InBetrieb AND Betriebsparameter.Boxen[5].Ventilator2));
	fbMinutenVentBox5.sekTick := sekTick;
	fbMinutenVentBox5.Minuten := ADR(hmiNutzungsdaten.Trocknungsbilanz.VentMinutenBox5);
	fbMinutenVentBox5();

	fbStundenVentBox5.Minuten := ADR(hmiNutzungsdaten.Trocknungsbilanz.VentMinutenBox5);
	fbStundenVentBox5.Stunden := ADR(hmiNutzungsdaten.Trocknungsbilanz.VentStundenBox5);
	fbStundenVentBox5();

	//Betrieb mit Luftaufbereitung
	fbMinutenLuftaufbBox5.Aktiv := Boxen.Box5Out.BoxBereit AND (((diBetriebsmldgKompressorModul1 OR diEntfeuchterFremdInBetrieb)  AND Betriebsparameter.Boxen[5].Luftentfeuchter) OR
	(diScheitholzofenInBetrieb AND Betriebsparameter.Boxen[5].Scheitholzofen) OR (doHeizregisterEin AND Betriebsparameter.Boxen[5].Heizregister) OR
	(Aktoren.Warmluftofen.WarmluftofenAktiv AND Betriebsparameter.Boxen[5].Warmluftofen)) ;
	fbMinutenLuftaufbBox5.sekTick := sekTick;
	fbMinutenLuftaufbBox5.Minuten := ADR(hmiNutzungsdaten.Trocknungsbilanz.LuftaufbMinutenBox5);
	fbMinutenLuftaufbBox5();

	fbStundenLuftaufbBox5.Minuten := ADR(hmiNutzungsdaten.Trocknungsbilanz.LuftaufbMinutenBox5);
	fbStundenLuftaufbBox5.Stunden := ADR(hmiNutzungsdaten.Trocknungsbilanz.LuftaufbStundenBox5);
	fbStundenLuftaufbBox5();

	//Box 6
	//*******************************************************************************************************************************

	//Gesamt
	fbMinutenBox6.Aktiv		:= Boxen.Box6Out.BoxBereit;
	fbMinutenBox6.sekTick	:= sekTick;
	fbMinutenBox6.Minuten	:= ADR(hmiNutzungsdaten.Bst.Box6Min);
	fbMinutenBox6();

	fbStundenBox6.Minuten	:= ADR(hmiNutzungsdaten.Bst.Box6Min);
	fbStundenBox6.Stunden	:= ADR(hmiNutzungsdaten.Bst.Box6Std);
	fbStundenBox6();

	//Ventilatorbetrieb
	fbMinutenVentBox6.Aktiv := Boxen.Box6Out.BoxBereit AND ((diVentilator1InBetrieb AND Betriebsparameter.Boxen[6].Ventilator1) OR
	(diVentilator2InBetrieb AND Betriebsparameter.Boxen[6].Ventilator2));
	fbMinutenVentBox6.sekTick := sekTick;
	fbMinutenVentBox6.Minuten := ADR(hmiNutzungsdaten.Trocknungsbilanz.VentMinutenBox6);
	fbMinutenVentBox6();

	fbStundenVentBox6.Minuten := ADR(hmiNutzungsdaten.Trocknungsbilanz.VentMinutenBox6);
	fbStundenVentBox6.Stunden := ADR(hmiNutzungsdaten.Trocknungsbilanz.VentStundenBox6);
	fbStundenVentBox6();

	//Betrieb mit Luftaufbereitung
	fbMinutenLuftaufbBox6.Aktiv := Boxen.Box6Out.BoxBereit AND (((diBetriebsmldgKompressorModul1 OR diEntfeuchterFremdInBetrieb)  AND Betriebsparameter.Boxen[6].Luftentfeuchter) OR
	(diScheitholzofenInBetrieb AND Betriebsparameter.Boxen[6].Scheitholzofen) OR (doHeizregisterEin AND Betriebsparameter.Boxen[6].Heizregister) OR
	(Aktoren.Warmluftofen.WarmluftofenAktiv AND Betriebsparameter.Boxen[6].Warmluftofen)) ;
	fbMinutenLuftaufbBox6.sekTick := sekTick;
	fbMinutenLuftaufbBox6.Minuten := ADR(hmiNutzungsdaten.Trocknungsbilanz.LuftaufbMinutenBox6);
	fbMinutenLuftaufbBox6();

	fbStundenLuftaufbBox6.Minuten := ADR(hmiNutzungsdaten.Trocknungsbilanz.LuftaufbMinutenBox6);
	fbStundenLuftaufbBox6.Stunden := ADR(hmiNutzungsdaten.Trocknungsbilanz.LuftaufbStundenBox6);
	fbStundenLuftaufbBox6();

	//======================================================================================================================================================
	//Restlaufzeiten von Boxen im Intervall- oder Nachtrocknungsbetrieb ermitteln
	//======================================================================================================================================================

	//Restzeiten Box 1
	fbRestzeitBox1.AktuelleMinute	:= Echtzeit.Minute;
	fbRestzeitBox1.AktuelleStunde	:= Echtzeit.Stunde;
	fbRestzeitBox1.Freigabe			:= Betriebsparameter.Boxen[1].IntervallbetriebEin OR Betriebsparameter.Boxen[1].NachtrocknungEin;
	IF Betriebsparameter.Boxen[1].IntervallbetriebEin THEN
		fbRestzeitBox1.ZeitfensterIn := ADR(Betriebsparameter.Boxen[1].IntervallbetriebZeiten);
	ELSE
		fbRestzeitBox1.ZeitfensterIn := ADR(Betriebsparameter.Boxen[1].NachtrocknungZeiten);
	END_IF
	fbRestzeitBox1();

	gStatusAnlage.RestlaufzeitenBoxen.Box1Minuten	:= fbRestzeitBox1.RestzeitMinutenOut;
	gStatusAnlage.RestlaufzeitenBoxen.Box1Stunden	:= fbRestzeitBox1.RestzeitStundenOut;

	//Restzeiten Box 2
	fbRestzeitBox2.AktuelleMinute	:= Echtzeit.Minute;
	fbRestzeitBox2.AktuelleStunde	:= Echtzeit.Stunde;
	fbRestzeitBox2.Freigabe			:= Betriebsparameter.Boxen[2].IntervallbetriebEin OR Betriebsparameter.Boxen[2].NachtrocknungEin;
	IF Betriebsparameter.Boxen[2].IntervallbetriebEin THEN
		fbRestzeitBox2.ZeitfensterIn := ADR(Betriebsparameter.Boxen[2].IntervallbetriebZeiten);
	ELSE
		fbRestzeitBox2.ZeitfensterIn := ADR(Betriebsparameter.Boxen[2].NachtrocknungZeiten);
	END_IF
	fbRestzeitBox2();

	gStatusAnlage.RestlaufzeitenBoxen.Box2Minuten	:= fbRestzeitBox2.RestzeitMinutenOut;
	gStatusAnlage.RestlaufzeitenBoxen.Box2Stunden	:= fbRestzeitBox2.RestzeitStundenOut;

	//Restzeiten Box 3
	fbRestzeitBox3.AktuelleMinute	:= Echtzeit.Minute;
	fbRestzeitBox3.AktuelleStunde	:= Echtzeit.Stunde;
	fbRestzeitBox3.Freigabe			:= Betriebsparameter.Boxen[3].IntervallbetriebEin OR Betriebsparameter.Boxen[3].NachtrocknungEin;
	IF Betriebsparameter.Boxen[3].IntervallbetriebEin THEN
		fbRestzeitBox3.ZeitfensterIn := ADR(Betriebsparameter.Boxen[3].IntervallbetriebZeiten);
	ELSE
		fbRestzeitBox3.ZeitfensterIn := ADR(Betriebsparameter.Boxen[3].NachtrocknungZeiten);
	END_IF
	fbRestzeitBox3();

	gStatusAnlage.RestlaufzeitenBoxen.Box3Minuten	:= fbRestzeitBox3.RestzeitMinutenOut;
	gStatusAnlage.RestlaufzeitenBoxen.Box3Stunden	:= fbRestzeitBox3.RestzeitStundenOut;

	//Restzeiten Box 4
	fbRestzeitBox4.AktuelleMinute	:= Echtzeit.Minute;
	fbRestzeitBox4.AktuelleStunde	:= Echtzeit.Stunde;
	fbRestzeitBox4.Freigabe			:= Betriebsparameter.Boxen[4].IntervallbetriebEin OR Betriebsparameter.Boxen[4].NachtrocknungEin;
	IF Betriebsparameter.Boxen[4].IntervallbetriebEin THEN
		fbRestzeitBox4.ZeitfensterIn := ADR(Betriebsparameter.Boxen[4].IntervallbetriebZeiten);
	ELSE
		fbRestzeitBox4.ZeitfensterIn := ADR(Betriebsparameter.Boxen[4].NachtrocknungZeiten);
	END_IF
	fbRestzeitBox4();

	gStatusAnlage.RestlaufzeitenBoxen.Box4Minuten	:= fbRestzeitBox4.RestzeitMinutenOut;
	gStatusAnlage.RestlaufzeitenBoxen.Box4Stunden	:= fbRestzeitBox4.RestzeitStundenOut;

	//Restzeiten Box 5
	fbRestzeitBox5.AktuelleMinute	:= Echtzeit.Minute;
	fbRestzeitBox5.AktuelleStunde	:= Echtzeit.Stunde;
	fbRestzeitBox5.Freigabe			:= Betriebsparameter.Boxen[5].IntervallbetriebEin OR Betriebsparameter.Boxen[5].NachtrocknungEin;
	IF Betriebsparameter.Boxen[5].IntervallbetriebEin THEN
		fbRestzeitBox5.ZeitfensterIn := ADR(Betriebsparameter.Boxen[5].IntervallbetriebZeiten);
	ELSE
		fbRestzeitBox5.ZeitfensterIn := ADR(Betriebsparameter.Boxen[5].NachtrocknungZeiten);
	END_IF
	fbRestzeitBox5();

	gStatusAnlage.RestlaufzeitenBoxen.Box5Minuten	:= fbRestzeitBox5.RestzeitMinutenOut;
	gStatusAnlage.RestlaufzeitenBoxen.Box5Stunden	:= fbRestzeitBox5.RestzeitStundenOut;

	//Restzeiten Box 6
	fbRestzeitBox6.AktuelleMinute	:= Echtzeit.Minute;
	fbRestzeitBox6.AktuelleStunde	:= Echtzeit.Stunde;
	fbRestzeitBox6.Freigabe			:= Betriebsparameter.Boxen[6].IntervallbetriebEin OR Betriebsparameter.Boxen[6].NachtrocknungEin;
	IF Betriebsparameter.Boxen[6].IntervallbetriebEin THEN
		fbRestzeitBox6.ZeitfensterIn := ADR(Betriebsparameter.Boxen[6].IntervallbetriebZeiten);
	ELSE
		fbRestzeitBox6.ZeitfensterIn := ADR(Betriebsparameter.Boxen[6].NachtrocknungZeiten);
	END_IF
	fbRestzeitBox6();

	gStatusAnlage.RestlaufzeitenBoxen.Box6Minuten	:= fbRestzeitBox6.RestzeitMinutenOut;
	gStatusAnlage.RestlaufzeitenBoxen.Box6Stunden	:= fbRestzeitBox6.RestzeitStundenOut;

	//======================================================================================================================================================
	//Serviceintervalle
	//======================================================================================================================================================

	hmiParameter.Servicebereich.KontrollintervallUhrzeit	:= 200000;
	//Kontrolle Uhrzeit
	fbSrvcUhrzeit.Aktiv				:= TRUE;
	fbSrvcUhrzeit.Tick				:= minTick;
	fbSrvcUhrzeit.ZeitBisSrvc		:= ADR(hmiNutzungsdaten.Serviceintervalle.RestzeitKontrolleUhrzeit);
	fbSrvcUhrzeit.SrvcIntervall		:= Betriebsparameter.Servicebereich.KontrollintervallUhrzeit;
	fbSrvcUhrzeit.SrvcReset			:= hmiButtons.ResetServiceUhrzeit;
	fbSrvcUhrzeit();
	hmiNutzungsdaten.Serviceintervalle.KontrolleUhrzeitErforderlich	:= fbSrvcUhrzeit.SrvcErforderl;

	IF (hmiButtons.ResetServiceUhrzeit) THEN
	hmiButtons.ResetServiceUhrzeit	:= FALSE;
	END_IF

	TON_ResetInit(IN:= TRUE, PT:= T#1s);
	initOk	:= TON_ResetInit.Q;

END_PROGRAM
```

#### Nutzung.var - Lokale Variablen
```iecst
(*============================================================================================================================================*)
(*======================================== FUNKTIONSBAUSTEINE FÜR ZEITTICKS =================================================================*)
VAR
	fbLascoZdxx_0 : fbLascoZdxx;
	fbLascoZdxx_1 : fbLascoZdxx;
	fbLascoZdxx_2 : fbLascoZdxx;
	fbLascoZdxx_3 : fbLascoZdxx;
	fbLascoZdxx_4 : fbLascoZdxx;
END_VAR
(*============================================================================================================================================*)
(*===================================================== ZEITTICKS==============================================================================*)
VAR
	sekTick : BOOL;
	minTick : BOOL;
	tagTick : BOOL;
	monatTick : BOOL;
	jahrTick : BOOL;
END_VAR
(*============================================================================================================================================*)
(*====================================== FUNKTIONSBAUSTEINE BETRIEBSSTUNDEN GESAMT=======================================================*)
VAR
	fbMinutenUmluftbetrGes : fbLascoBmin;
	fbStundenUmluftbetrGes : fbLascoStdMin;
	fbMinutenFrischluftbetrGes : fbLascoBmin;
	fbStundenFrischluftbetrGes : fbLascoStdMin;
	fbMinutenAbluftventGes : fbLascoBmin;
	fbStundenAbluftventGes : fbLascoStdMin;
	fbMinutenVentilator1Ges : fbLascoBmin;
	fbStundenVentilator1Ges : fbLascoStdMin;
	fbMinutenVentilator2Ges : fbLascoBmin;
	fbStundenVentilator2Ges : fbLascoStdMin;
	fbMinutenOelsumpfhGes : fbLascoBmin;
	fbStundenOelsumpfhGes : fbLascoStdMin;
	fbMinutenKompressor1Ges : fbLascoBmin;
	fbStundenKompressor1Ges : fbLascoStdMin;
	fbMinutenKompressor2Ges : fbLascoBmin;
	fbStundenKompressor2Ges : fbLascoStdMin;
	fbMinutenAbtauung1Ges : fbLascoBmin;
	fbStundenAbtauung1Ges : fbLascoStdMin;
	fbMinutenAbtauung2Ges : fbLascoBmin;
	fbStundenAbtauung2Ges : fbLascoStdMin;
	fbMinutenWarmluftofenGes : fbLascoBmin;
	fbStundenWarmluftofenGes : fbLascoStdMin;
	fbMinutenScheitholzofenGes : fbLascoBmin;
	fbStundenScheitholzofenGes : fbLascoStdMin;
	fbMinutenHeizregisterGes : fbLascoBmin;
	fbStundenHeizregisterGes : fbLascoStdMin;
	fbMinutenBox1Ges : fbLascoBmin;
	fbStundenBox1Ges : fbLascoStdMin;
	fbMinutenBox2Ges : fbLascoBmin;
	fbStundenBox2Ges : fbLascoStdMin;
	fbMinutenBox3Ges : fbLascoBmin;
	fbStundenBox3Ges : fbLascoStdMin;
	fbMinutenBox4Ges : fbLascoBmin;
	fbStundenBox4Ges : fbLascoStdMin;
	fbMinutenBox5Ges : fbLascoBmin;
	fbStundenBox5Ges : fbLascoStdMin;
	fbMinutenBox6Ges : fbLascoBmin;
	fbStundenBox6Ges : fbLascoStdMin;
END_VAR
(*====================================== FUNKTIONSBAUSTEINE BETRIEBSSTUNDEN ===============================================================*)
(*============================================================================================================================================*)
VAR
	fbMinutenUmluftbetr : fbLascoBmin;
	fbStundenUmluftbetr : fbLascoStdMin;
	fbMinutenFrischluftbetr : fbLascoBmin;
	fbStundenFrischluftbetr : fbLascoStdMin;
	fbMinutenAbluftvent : fbLascoBmin;
	fbStundenAbluftvent : fbLascoStdMin;
	fbMinutenVentilator1 : fbLascoBmin;
	fbStundenVentilator1 : fbLascoStdMin;
	fbMinutenVentilator2 : fbLascoBmin;
	fbStundenVentilator2 : fbLascoStdMin;
	fbMinutenOelsumpfh : fbLascoBmin;
	fbStundenOelsumpfh : fbLascoStdMin;
	fbMinutenKompressor1 : fbLascoBmin;
	fbStundenKompressor1 : fbLascoStdMin;
	fbMinutenKompressor2 : fbLascoBmin;
	fbStundenKompressor2 : fbLascoStdMin;
	fbMinutenAbtauung1 : fbLascoBmin;
	fbStundenAbtauung1 : fbLascoStdMin;
	fbMinutenAbtauung2 : fbLascoBmin;
	fbStundenAbtauung2 : fbLascoStdMin;
	fbMinutenWarmluftofen : fbLascoBmin;
	fbStundenWarmluftofen : fbLascoStdMin;
	fbMinutenScheitholzofen : fbLascoBmin;
	fbStundenScheitholzofen : fbLascoStdMin;
	fbMinutenHeizregister : fbLascoBmin;
	fbStundenHeizregister : fbLascoStdMin;
	fbMinutenBox1 : fbLascoBmin;
	fbStundenBox1 : fbLascoStdMin;
	fbMinutenVentBox1 : fbLascoBmin;
	fbStundenVentBox1 : fbLascoStdMin;
	fbMinutenLuftaufbBox1 : fbLascoBmin;
	fbStundenLuftaufbBox1 : fbLascoStdMin;
	fbMinutenVentBox2 : fbLascoBmin;
	fbStundenVentBox2 : fbLascoStdMin;
	fbMinutenLuftaufbBox2 : fbLascoBmin;
	fbStundenLuftaufbBox2 : fbLascoStdMin;
	fbMinutenVentBox3 : fbLascoBmin;
	fbStundenVentBox3 : fbLascoStdMin;
	fbMinutenLuftaufbBox3 : fbLascoBmin;
	fbStundenLuftaufbBox3 : fbLascoStdMin;
	fbMinutenVentBox4 : fbLascoBmin;
	fbStundenVentBox4 : fbLascoStdMin;
	fbMinutenLuftaufbBox4 : fbLascoBmin;
	fbStundenLuftaufbBox4 : fbLascoStdMin;
	fbMinutenVentBox5 : fbLascoBmin;
	fbStundenVentBox5 : fbLascoStdMin;
	fbMinutenLuftaufbBox5 : fbLascoBmin;
	fbStundenLuftaufbBox5 : fbLascoStdMin;
	fbMinutenVentBox6 : fbLascoBmin;
	fbStundenVentBox6 : fbLascoStdMin;
	fbMinutenLuftaufbBox6 : fbLascoBmin;
	fbStundenLuftaufbBox6 : fbLascoStdMin;
	fbMinutenBox2 : fbLascoBmin;
	fbStundenBox2 : fbLascoStdMin;
	fbMinutenBox3 : fbLascoBmin;
	fbStundenBox3 : fbLascoStdMin;
	fbMinutenBox4 : fbLascoBmin;
	fbStundenBox4 : fbLascoStdMin;
	fbMinutenBox5 : fbLascoBmin;
	fbStundenBox5 : fbLascoStdMin;
	fbMinutenBox6 : fbLascoBmin;
	fbStundenBox6 : fbLascoStdMin;
END_VAR
(*============================================================================================================================================*)
(*====================================== FUNKTIONSBAUSTEINE SERVICEINTERVALLE==============================================================*)
VAR
	fbSrvcUhrzeit : fbLascoSrvcInterv;
	DTGetTime_0 : DTGetTime;
	loc_UhrzeitAktuellUdint : UDINT;
	TON_MinLaufzeitOelsumpfh : TON;
	loc_MinLaufzeitOelsumpf : UDINT;
	TON_ResetInit : TON;
	loc_UhrzeitMEM_Udint : UDINT;
	initOk : BOOL;
	stateEntry : BOOL;
	loc_ZeitStromausfall : UDINT;
END_VAR
(*============================================================================================================================================*)
(*====================================== FUNKTIONSBAUSTEINE RESTZEITEN BOXEN ============================================================*)
VAR
	fbRestzeitBox1 : {REDUND_UNREPLICABLE} fbRestzeit;
	fbRestzeitBox2 : {REDUND_UNREPLICABLE} fbRestzeit;
	fbRestzeitBox3 : {REDUND_UNREPLICABLE} fbRestzeit;
	fbRestzeitBox4 : {REDUND_UNREPLICABLE} fbRestzeit;
	fbRestzeitBox5 : {REDUND_UNREPLICABLE} fbRestzeit;
	fbRestzeitBox6 : {REDUND_UNREPLICABLE} fbRestzeit;
END_VAR
```

### Program Logical/Util/System (IEC) - Ethernet konfigurieren

#### System.st - Zyklischer Code
```iecst
(********************************************************************
 * COPYRIGHT -- LASCO Heu- und Forsttechnik GmbH
 ********************************************************************
 * Programm: System
 * Datei: System.st
 * Autor: Rudolf Lachner
 * Erstellt: 16. Januar 2014
 ********************************************************************
 * Implementierung des Programms System
 ********************************************************************)

PROGRAM _CYCLIC

	//Ticks generieren
	//****************
	fbLascoZdxx_0(IN 	:= hmiStatus.CurPage);
	bildTick			:= fbLascoZdxx_0.Q;
	fbLascoZdxx_1(IN	:= Echtzeit.Sekunde);
	sekTick				:= fbLascoZdxx_1.Q;

	//Name der Schnittstelle
	strcpy(ADR(Device), ADR('IF3'));

	//Konfiguration der IP- Adresse
	//*****************************

	IF (EDGEPOS(hmiButtons.IpParameterSetzen)) THEN
		Nutzungsdaten.Allgemein.SetEthernetOk	:= FALSE;
		CfgSetIPAddr_status         	:= ERR_FUB_BUSY;
		CfgSetDefaultGateway_status 	:= ERR_FUB_BUSY;
		CfgSetSubnetMask_status     	:= ERR_FUB_BUSY;
		CfgSetHostName_status       	:= ERR_FUB_BUSY;
	END_IF

	//Ethernetparameter setzen
	//************************
	IF (hmiButtons.IpParameterSetzen) THEN

		//IP- Adresse bei Init
		IF (CfgSetIPAddr_status <> 0) THEN
			CfgSetIPAddr_0(enable 	:= TRUE, pDevice := ADR(Device), pIPAddr := ADR(Betriebsparameter.Allgemein.IPAdresse) , Option := 1);
			CfgSetIPAddr_status		:= CfgSetIPAddr_0.status;
		END_IF

		//Subnet Maske
		IF (CfgSetIPAddr_status = 0) AND (CfgSetSubnetMask_status <> 0) THEN
			CfgSetSubnetMask_0(enable 	:= TRUE, pDevice := ADR(Device), pSubnetMask := ADR(Betriebsparameter.Allgemein.SubnetMask), Option := 1);
			CfgSetSubnetMask_status		:= CfgSetSubnetMask_0.status;
		END_IF

		//Default Gateway
		IF (CfgSetIPAddr_status = 0) AND (CfgSetSubnetMask_status = 0) AND (CfgSetDefaultGateway_status <> 0) THEN
			CfgSetDefaultGateway_0(enable 	:= TRUE, pDevice := ADR(Device), pGateway := ADR(Betriebsparameter.Allgemein.DefaultGateway), Option := 1);
			CfgSetDefaultGateway_status		:= CfgSetDefaultGateway_0.status;
		END_IF

		//Host- Name
		IF (CfgSetHostName_status <> 0) THEN
			CfgSetHostName_0(enable := TRUE, pHostName := ADR(Betriebsparameter.Allgemein.HostName), Option := 1);
			CfgSetHostName_status	:= CfgSetHostName_0.status;
		END_IF

		//Konfiguration abschließen
		IF (CfgSetIPAddr_status = 0) AND (CfgSetDefaultGateway_status = 0) AND (CfgSetSubnetMask_status = 0) AND (CfgSetSubnetMask_status = 0) THEN
			hmiButtons.IpParameterSetzen     				:= FALSE;
			Nutzungsdaten.Allgemein.SetEthernetOk		:= TRUE;
		END_IF
	END_IF

	(*
	//Ethernetparameter auslesen
	//**************************
	IF (hmiStatus.hmiCurPage = _650_SYS) AND (bildTick) THEN
		loc_GetEthernet 			:= TRUE;
		CfgGetIPAddr_status         := ERR_FUB_BUSY;
		CfgGetDefaultGateway_status := ERR_FUB_BUSY;
		CfgGetSubnetMask_status     := ERR_FUB_BUSY;
		CfgGetHostName_status       := ERR_FUB_BUSY;
	END_IF

	TON_10ms_0(IN := loc_GetEthernet, PT := 2 * 100);

	IF loc_GetEthernet THEN

		hmiActions.cmdSetIpAddress	:= FALSE;

		//IP- Adresse
		IF CfgGetIPAddr_status <> 0 THEN
			CfgGetIPAddr_0(enable 	:= TRUE, pDevice := ADR(Device), pIPAddr := ADR(Betriebsparameter.Allgemein.IPAdresse), Len := INT_TO_USINT(LEN(Betriebsparameter.Allgemein.IPAdresse) + 1));
			CfgGetIPAddr_status		:= CfgGetIPAddr_0.status;
		END_IF

		//Subnet Maske
		IF CfgGetSubnetMask_status <> 0 THEN
			CfgGetSubnetMask_0(enable 	:= TRUE, pDevice := ADR(Device), pSubnetMask := ADR(Betriebsparameter.Allgemein.SubnetMask), Len := INT_TO_USINT(LEN(Betriebsparameter.Allgemein.SubnetMask) + 1));
			CfgGetSubnetMask_status		:= CfgGetSubnetMask_0.status;
		END_IF

		//Default Gateway
		IF CfgGetDefaultGateway_status <> 0 THEN
			CfgGetDefaultGateway_0(enable 	:= TRUE, pDevice := ADR(Device), pGateway := ADR(Betriebsparameter.Allgemein.DefaultGateway), Len := INT_TO_USINT(LEN(Betriebsparameter.Allgemein.DefaultGateway) + 1));
			CfgGetDefaultGateway_status		:= CfgGetDefaultGateway_0.status;
		END_IF

		//Host Name
		IF CfgGetHostName_status <> 0 THEN
			CfgGetHostName_0(enable := TRUE, pHostName := ADR(Betriebsparameter.Allgemein.HostName), Len := INT_TO_USINT(LEN(Betriebsparameter.Allgemein.HostName) + 1));
			CfgGetHostName_status	:= CfgGetHostName_0.status;
		END_IF

		IF (CfgGetIPAddr_status = 0) AND (CfgGetDefaultGateway_status = 0) AND (CfgGetSubnetMask_status = 0) AND (CfgGetHostName_status = 0) THEN
			loc_GetEthernet		:= FALSE;
		ELSIF TON_10ms_0.Q THEN
			loc_GetEthernet	:= FALSE;
		END_IF
	END_IF*)

END_PROGRAM
```

#### System.var - Lokale Variablen
```iecst
(*============================================================================================================================================*)
(*======================================== FUNKTIONSBAUSTEINE FÜR TICKS =====================================================================*)
VAR
	fbLascoZdxx_0 : fbLascoZdxx;
	fbLascoZdxx_1 : fbLascoZdxx;
END_VAR
(*============================================================================================================================================*)
(*====================================================== TICKS ================================================================================*)
VAR
	bildTick : BOOL;
	sekTick : BOOL;
END_VAR
(*============================================================================================================================================*)
(*====================================================== ANDERE ==============================================================================*)
VAR
	Device : STRING[16];
	loc_GetEthernet : BOOL;
	TON_10ms_0 : TON_10ms;
END_VAR
(*============================================================================================================================================*)
(*======================================== FUNKTIONSBAUSTEINE SETZEN ETHERNET=============================================================*)
VAR
	CfgSetIPAddr_status : UINT;
	CfgSetDefaultGateway_status : UINT;
	CfgSetSubnetMask_status : UINT;
	CfgSetHostName_status : UINT;
	CfgSetIPAddr_0 : CfgSetIPAddr;
	CfgSetSubnetMask_0 : CfgSetSubnetMask;
	CfgSetDefaultGateway_0 : CfgSetDefaultGateway;
	CfgSetHostName_0 : CfgSetHostName;
END_VAR
(*============================================================================================================================================*)
(*======================================== FUNKTIONSBAUSTEINE LESEN ETHERNET===============================================================*)
VAR
	CfgGetIPAddr_status : UINT;
	CfgGetSubnetMask_status : UINT;
	CfgGetDefaultGateway_status : UINT;
	CfgGetHostName_status : UINT;
	CfgGetIPAddr_0 : CfgGetIPAddr;
	CfgGetSubnetMask_0 : CfgGetSubnetMask;
	CfgGetDefaultGateway_0 : CfgGetDefaultGateway;
	CfgGetHostName_0 : CfgGetHostName;
END_VAR
```

### Program Logical/Util/mappPara (IEC) - Parametersicherung in XML-Files

#### Main.st - Init, cyclic, exit code
```iecst
PROGRAM _INIT

	hmiParameter;
	MpRecipeXml_0.Enable		:= FALSE;
	MpRecipeXml_0();
	MpRecipeRegPar_0.Enable		:= FALSE;
	MpRecipeRegPar_0();
	MpRecipeUI_0.Enable			:= FALSE;
	MpRecipeUI_0();
	FileCopy_0.enable			:= FALSE;
	FileCopy_0();

	hmiStatus.ParameterFileNameAufUsb	:= 'FileNameAufUsb';

	//Standardparametersatz laden, wenn keine Parameter vorhanden (neues Display)
	IF (NOT Betriebsparameter.Allgemein.ParameterVorhanden) THEN
		gWerksparameterLaden	:= TRUE;
	END_IF

END_PROGRAM

PROGRAM _CYCLIC

	//Parametersatz-Verwaltung mittels mapp-Service im XML-Dateiformat
	//================================================================
	//Parametersätze können wahlweise von der USER-Partition am Display,
	//oder von einem USB-Stick geladen werden.

	//Schreibschutz für StandardParametersätze
	IF (UIConnect.New.FileName = '207Werk') OR (UIConnect.New.FileName = '307Werk') OR (UIConnect.New.FileName = '407Werk') OR (UIConnect.New.FileName = '407PlusWerk') OR (UIConnect.New.FileName = '304Werk') OR
		(UIConnect.New.FileName = 'HB4000Werk') OR (UIConnect.New.FileName = 'HB3000Werk') OR (FileNameFromUSB = '207Werk') OR (FileNameFromUSB = '307Werk') OR (FileNameFromUSB = '407Werk') OR
		(FileNameFromUSB = '407PlusWerk') OR (FileNameFromUSB = '304Werk') OR (FileNameFromUSB = 'HB4000Werk') OR (FileNameFromUSB = 'HB3000Werk') THEN
		loc_LockNewFile	:= TRUE;
	ELSE
		loc_LockNewFile	:= FALSE;
	END_IF

	//Schrittschaltwerk Parametersicherung
	//************************************

	CASE step OF

		//**********************************************************************************************************
		//DATEIVERWALTUNG VON BENUTZERPARTITION F:\
		0:

			//*** state entry ***
			IF stateEntry THEN
				stateEntry	:= FALSE;
				MpRecipeXml_0.Enable		:= FALSE;
				MpRecipeXml_0.ErrorReset	:= FALSE;
				MpRecipeXml_0();
				MpRecipeRegPar_0.Enable		:= FALSE;
				MpRecipeRegPar_0.ErrorReset	:= FALSE;
				MpRecipeRegPar_0();
				MpRecipeUI_0.Enable			:= FALSE;
				MpRecipeUI_0.ErrorReset		:= FALSE;
				MpRecipeUI_0();
				hmiButtons.ParameterAufUsbKopieren := FALSE;
				hmiButtons.ParameterVonUsbLaden := FALSE;
			END_IF

			//*** state during ***
			MpRecipeXml_0.Enable		:= TRUE;
			MpRecipeXml_0.MpLink		:= ADR(gMappRecipeLink);
			MpRecipeXml_0.DeviceName	:= ADR('CF');
			MpRecipeXml_0.FileName		:= ADR('407Werk');
			MpRecipeXml_0();

			MpRecipeRegPar_0.MpLink		:= ADR(gMappRecipeLink);
			MpRecipeRegPar_0.Enable		:= TRUE;
			MpRecipeRegPar_0.PVName		:= ADR('hmiParameter');
			MpRecipeRegPar_0();

			MpRecipeUI_0.MpLink			:= ADR(gMappRecipeLink);
			MpRecipeUI_0.Enable			:= TRUE;
			MpRecipeUI_0.UISetup		:= UISetup;
			MpRecipeUI_0.UIConnect		:= ADR(UIConnect);
			MpRecipeUI_0();

			//*** state exit ***
			//Parametersatz von USB laden
			IF hmiButtons.ParameterVonUsbLaden THEN
				stateEntry	:= TRUE;
				step		:= 1;
			//Ausgewählten Parametersatz auf USB-Stick kopieren
			ELSIF hmiButtons.ParameterAufUsbKopieren THEN
				stateEntry	:= TRUE;
				step		:= 3;
			//Keine Parameter vorhanden -> Werksparameter laden
			ELSIF gWerksparameterLaden THEN
				stateEntry	:= TRUE;
				step		:= 4;
				//Fehler -> Reset
			ELSIF MpRecipeXml_0.Error OR MpRecipeRegPar_0.Error OR MpRecipeUI_0.Error THEN
				stateEntry	:= TRUE;
				step		:= 255;
			END_IF

		//**********************************************************************************************************
		//DATEI VON USB-STICK LADEN
		1:

			//*** state entry ***
			IF stateEntry THEN
				stateEntry	:= FALSE;
				MpRecipeXml_0.Enable		:= FALSE;
				MpRecipeXml_0();
				MpRecipeRegPar_0.Enable		:= FALSE;
				MpRecipeRegPar_0();
				MpRecipeUI_0.Enable			:= FALSE;
				MpRecipeUI_0();
			END_IF

			//*** state during ***
			MpRecipeXml_0.Enable		:= TRUE;

			MpRecipeXml_0.MpLink		:= ADR(gMappRecipeLink);
			MpRecipeXml_0.DeviceName	:= ADR('usb_device');
			MpRecipeXml_0.FileName		:= ADR(hmiStatus.ParameterFileNameAufUsb);
			MpRecipeXml_0();

			MpRecipeRegPar_0.MpLink		:= ADR(gMappRecipeLink);
			MpRecipeRegPar_0.Enable		:= TRUE;
			MpRecipeRegPar_0.PVName		:= ADR('hmiParameter');
			MpRecipeRegPar_0();

			MpRecipeXml_0.Load			:= TRUE;

			//*** state exit ***
			//Parametersatz von USB fertig geladen -> Neuen Parametersatz mit selben Namen auf F:\ ablegen
			IF MpRecipeXml_0.CommandDone THEN
				MpRecipeXml_0.Load		:= FALSE;
				stateEntry				:= TRUE;
				step					:= 2;
			//Fehler -> Reset
			ELSIF MpRecipeXml_0.Error OR MpRecipeRegPar_0.Error OR MpRecipeUI_0.Error THEN
				stateEntry	:= TRUE;
				step		:= 255;
			END_IF

		//**********************************************************************************************************
		//DATEI VON USB-STICK AUF BENUTZERPARTITION SPEICHERN
		2:
			//*** state entry ***
			IF stateEntry THEN
				stateEntry	:= FALSE;
				MpRecipeXml_0.Enable		:= FALSE;
				MpRecipeXml_0();
				MpRecipeRegPar_0.Enable		:= FALSE;
				MpRecipeRegPar_0();
				MpRecipeUI_0.Enable			:= FALSE;
				MpRecipeUI_0();
			END_IF

			MpRecipeXml_0.Enable		:= TRUE;
			MpRecipeXml_0.MpLink		:= ADR(gMappRecipeLink);
			MpRecipeXml_0.DeviceName	:= ADR('CF');
			MpRecipeXml_0.FileName		:= ADR('407Werk');
			MpRecipeXml_0();

			MpRecipeRegPar_0.MpLink		:= ADR(gMappRecipeLink);
			MpRecipeRegPar_0.Enable		:= TRUE;
			MpRecipeRegPar_0.PVName		:= ADR('hmiParameter');
			MpRecipeRegPar_0();

			MpRecipeUI_0.MpLink			:= ADR(gMappRecipeLink);
			MpRecipeUI_0.Enable			:= TRUE;
			MpRecipeUI_0.UISetup		:= UISetup;
			MpRecipeUI_0.UIConnect		:= ADR(UIConnect);
			MpRecipeUI_0();

			UIConnect.New.FileName		:= hmiStatus.ParameterFileNameAufUsb;
			UIConnect.New.Create		:= TRUE;

			//*** state exit ***
			//Parametersatz abgespeichert
			IF MpRecipeXml_0.CommandDone THEN
				UIConnect.Recipe.Refresh	:= TRUE;
				stateEntry					:= TRUE;
				step						:= 0;
				//Fehler -> Reset
			ELSIF MpRecipeXml_0.Error OR MpRecipeRegPar_0.Error OR MpRecipeUI_0.Error THEN
				stateEntry	:= TRUE;
				step		:= 255;
			END_IF

		//**********************************************************************************************************
		//PARAMETERSATZ AUF USB-STICK KOPIEREN
		3:

			//*** state entry ***
			IF stateEntry THEN
				stateEntry	:= FALSE;
				MpRecipeXml_0.Enable		:= FALSE;
				MpRecipeXml_0();
				MpRecipeRegPar_0.Enable		:= FALSE;
				MpRecipeRegPar_0();
				MpRecipeUI_0.Enable			:= FALSE;
				MpRecipeUI_0();
				FileCopy_0.enable			:= FALSE;
				FileCopy_0();
			END_IF

			//*** state during ***
			loc_FileName	:= UIConnect.Recipe.List.Names[UIConnect.Recipe.List.SelectedIndex];

			FileCopy_0.enable 	:= TRUE;
			FileCopy_0.option	:= fiOVERWRITE;
			FileCopy_0.pDest	:= ADR(loc_FileName);
			FileCopy_0.pDestDev	:= ADR('usb_device');
			FileCopy_0.pSrc		:= ADR(loc_FileName);
			FileCopy_0.pSrcDev	:= ADR('CF');
			FileCopy_0();

			//*** state exit ***
			//Parametersatz auf USB kopiert
			IF FileCopy_0.status = 0 THEN
				stateEntry 	:= TRUE;
				step		:= 0;
			//Fehler
			ELSIF FileCopy_0.status <> ERR_FUB_BUSY THEN
				stateEntry	:= TRUE;
				step		:= 255;
			END_IF

		//**********************************************************************************************************
		//WERKSPARAMETER BEI NEUEM DISPLAY LADEN
		4:

			//*** state entry ***
			IF stateEntry THEN
				stateEntry	:= FALSE;
				MpRecipeXml_0.Enable		:= FALSE;
				MpRecipeXml_0();
				MpRecipeRegPar_0.Enable		:= FALSE;
				MpRecipeRegPar_0();
				MpRecipeUI_0.Enable			:= FALSE;
				MpRecipeUI_0();
				gWerksparameterLaden		:= FALSE;
			END_IF

			//*** state during ***
			MpRecipeXml_0.Enable		:= TRUE;

			MpRecipeXml_0.MpLink		:= ADR(gMappRecipeLink);
			MpRecipeXml_0.DeviceName	:= ADR('CF');
			IF hmiStatus.NameSteuerung = 0 THEN
				MpRecipeXml_0.FileName		:= ADR('407Werk');
			ELSIF hmiStatus.NameSteuerung = 1 THEN
				MpRecipeXml_0.FileName		:= ADR('407PlusWerk');
			ELSIF hmiStatus.NameSteuerung = 2 THEN
				MpRecipeXml_0.FileName		:= ADR('307Werk');
			ELSIF hmiStatus.NameSteuerung = 3 THEN
				MpRecipeXml_0.FileName		:= ADR('304Werk');
			ELSIF hmiStatus.NameSteuerung = 4 THEN
				MpRecipeXml_0.FileName		:= ADR('HB4000Werk');
			ELSIF hmiStatus.NameSteuerung = 5 THEN
				MpRecipeXml_0.FileName		:= ADR('HB3000Werk');
			ELSIF hmiStatus.NameSteuerung = 6 THEN
				MpRecipeXml_0.FileName		:= ADR('207Werk');
			END_IF
			MpRecipeXml_0();

			MpRecipeRegPar_0.MpLink		:= ADR(gMappRecipeLink);
			MpRecipeRegPar_0.Enable		:= TRUE;
			MpRecipeRegPar_0.PVName		:= ADR('hmiParameter');
			MpRecipeRegPar_0();

			MpRecipeXml_0.Load			:= TRUE;

			//*** state exit ***
			//Parametersatz geladen
			IF MpRecipeXml_0.CommandDone THEN
				MpRecipeXml_0.Load		:= FALSE;
				stateEntry				:= TRUE;
				step					:= 0;
			//Fehler -> Reset
			ELSIF MpRecipeXml_0.Error OR MpRecipeRegPar_0.Error OR MpRecipeUI_0.Error THEN
				stateEntry	:= TRUE;
				step		:= 255;
			END_IF

		//**********************************************************************************************************
		//FEHLER
		255:

			//*** state entry ***
			IF stateEntry THEN
				stateEntry	:= FALSE;
			END_IF

			MpRecipeXml_0.ErrorReset	:= TRUE;
			MpRecipeXml_0();

			MpRecipeRegPar_0.ErrorReset	:= TRUE;
			MpRecipeRegPar_0();

			MpRecipeUI_0.ErrorReset		:= TRUE;
			MpRecipeUI_0();

			step:= 0;
			stateEntry := TRUE;

	END_CASE

END_PROGRAM

PROGRAM _EXIT

	MpRecipeXml_0.Enable		:= FALSE;
	MpRecipeXml_0();
	MpRecipeRegPar_0.Enable		:= FALSE;
	MpRecipeRegPar_0();
	MpRecipeUI_0.Enable			:= FALSE;
	MpRecipeUI_0();

END_PROGRAM
```

#### Variables.var - Local variables
```iecst
VAR
	MpRecipeXml_0 : MpRecipeXml;
	MpRecipeRegPar_0 : MpRecipeRegPar;
	MpRecipeUI_0 : MpRecipeUI;
	stateEntry : BOOL := 0;
	FileNameFromUSB : STRING[80] := 'FileNameAufUSB';
	UISetup : MpRecipeUISetupType;
	UIConnect : MpRecipeUIConnectType := (New:=(FileName:='NeuerFileName'));
	step : USINT := 0;
	loc_LockNewFile : BOOL := 0;
	FileCopy_0 : {REDUND_UNREPLICABLE} FileCopy;
	loc_FileName : {REDUND_UNREPLICABLE} STRING[30];
END_VAR
```

### InputOutput.var
```iecst
(*Digitale Ausgänge (DO) ===================================================================================================================================================*)
VAR
	doVentilator1Ein : BOOL;
	doVentilator2Ein : BOOL;
	doTrocknungInBetrieb : BOOL;
	doFreigabeBox1 : BOOL;
	doFreigabeBox2 : BOOL;
	doTrocknungStoerung : BOOL;
	doWarmluftofenEin : BOOL;
	doHeizregisterEin : BOOL;
	doFreigabeBox3 : BOOL;
	doFreigabeBox4 : BOOL;
	doFreigabeBox5 : BOOL;
	doFreigabeBox6 : BOOL;
	doBrandschutzklappeAuf : BOOL;
	doAbluftventilatorEin : BOOL;
	doAbluftklappeFreigabe : BOOL;
	doAbluftklappeOeffnen : BOOL; (*Nur bei 3.04 in Verwendung*)
	doAbluftklappeSchliessen : BOOL; (*Nur bei 3.04 in Verwendung*)
	doUmluftklappe2Schliessen : BOOL; (*Nur bei 3.04 in Verwendung*)
	doUmluftklappe2Oeffnen : BOOL; (*Nur bei 3.04 in Verwendung*)
	doUmluftklappe1Schliessen : BOOL; (*Nur bei 3.04 in Verwendung*)
	doUmluftklappe1Oeffnen : BOOL; (*Nur bei 3.04 in Verwendung*)
	doUmluftklappe1Freigabe : BOOL;
	doUmluftklappe2Freigabe : BOOL;
	doNotstromaggregatEin : BOOL;
	doKompressorEinModul1 : BOOL;
	doKompressorEinModul2 : BOOL;
	doMagnetventilEinModul1 : BOOL;
	doMagnetventilEinModul2 : BOOL;
	doOelsumpfheizungEinModul1 : BOOL;
	doOelsumpfheizungEinModul2 : BOOL;
	doBypassklappeSchliessen : BOOL; (*Nur bei 3.04 in Verwendung*)
	doBypassklappeOeffnen : BOOL;
	doEntfFremdFreigabe : BOOL; (*Nur bei HB4000 in Verwendung*)
	doLuftentfeuchterStrombegrEin : BOOL; (*Nur bei HB4000 in Verwendung*)
END_VAR
(*Analoge Ausgänge (AO) =====================================================================================================================================================*)
VAR
	aoDrehzahlvorgVentilator1 : REAL;
	aoTemperaturvorgWarmluftofen : REAL;
	aoDrehzahlvorgVentilator2 : REAL;
	aoLeistungsvorgHeizregister : REAL;
	aoDrehzahlvorgAbluftventilator : REAL;
	aoDrehzahlvorgKompressorModul1 : REAL;
	aoDrehzahlvorgKompressorModul2 : REAL;
END_VAR
(*Analoge Eingänge (AI) =====================================================================================================================================================*)
VAR
	aiFrischluftTemperatur : REAL;
	aiFrischluftFeuchte : REAL;
	aiTrockenluftTemperatur : REAL;
	aiTrockenluftFeuchte : REAL;
	aiAbluftTemperatur : REAL;
	aiAbluftFeuchte : REAL;
	aiDachluftTemperatur : REAL;
	aiDachluftFeuchte : REAL;
	aiLuftgeschwindigkeit : REAL;
	aiDifferenzdruck : REAL;
	aiNiederdruckModul2 : REAL;
	aiNiederdruckModul1 : REAL;
	aiHochdruckModul2 : REAL;
	aiHochdruckModul1 : REAL;
	aiEintrittTemperatur : REAL;
	aiEintrittFeuchte : REAL;
	aiAustrittTemperatur : REAL;
	aiAustrittFeuchte : REAL;
END_VAR
(*Digitale Eingänge (DI) =====================================================================================================================================================*)
VAR
	di230VACIstOk : BOOL; (*Nur bei HB4000 in Verwendung*)
	diEntfeuchterFremdInBetrieb : BOOL; (*Nur bei HB4000 in Verwendung*)
	diEntfeuchterFremdStoerung : BOOL; (*Nur bei HB4000 in Verwendung*)
	diTasteTrocknungPausieren : BOOL; (*Nur bei HB4000 in Verwendung*)
	diDrehfeldIstKorrekt : BOOL; (*Nur bei 3.04 in Verwendung*)
	diVentilator1InBetrieb : BOOL;
	di24VDCinternIstOk : BOOL;
	diBox1Offen : BOOL;
	diBox1Geschl : BOOL;
	diBox2Offen : BOOL;
	diBox2Geschl : BOOL;
	diVentilator2InBetrieb : BOOL;
	diDrehzahlbegrVentilator1 : BOOL;
	diDrehzahlbegrVentilator2 : BOOL;
	diScheitholzofenInBetrieb : BOOL;
	diWarmluftofenInBetrieb : BOOL;
	diBox3Offen : BOOL;
	diBox3Geschl : BOOL;
	diBox4Offen : BOOL;
	diBox4Geschl : BOOL;
	diBox5Offen : BOOL;
	diBox5Geschl : BOOL;
	diBox6Offen : BOOL;
	diBox6Geschl : BOOL;
	diAbluftventInBetrieb : BOOL;
	diAbluftklappeOffen : BOOL;
	diAbluftklappeGeschl : BOOL;
	diUmschaltklappe1Offen : BOOL;
	diUmschaltklappe1Geschl : BOOL;
	diUmschaltklappe2Offen : BOOL;
	diUmschaltklappe2Geschl : BOOL;
	diNotstromaggregatInBetrieb : BOOL;
	diNiederdruckOkModul1 : BOOL;
	diNiederdruckOkModul2 : BOOL;
	diHochdruckOkModul1 : BOOL;
	diHochdruckOkModul2 : BOOL;
	diKopftempKompressorModul1 : BOOL;
	diKopftempKompressorModul2 : BOOL;
	diOeldruckKompressorModul1 : BOOL;
	diOeldruckKompressorModul2 : BOOL;
	diVollschutzKompressorModul1 : BOOL;
	diVollschutzKompressorModul2 : BOOL;
	diBetriebsmldgKompressorModul1 : BOOL;
	diBetriebsmldgKompressorModul2 : BOOL;
	diAnfEntfeuchterExtern : BOOL;
	diLeistungsvorgKompressorExtMod1 : BOOL;
	diBypassklappeGeschl : BOOL;
	diBypassklappeOffen : BOOL;
	diHeizregisterFrostschutz : BOOL;
END_VAR
(*Statuseingänge (DI) =====================================================================================================================================================*)
VAR
	diStatusNiederdruckMinMod1 : BOOL;
	diStatusNiederdruckMaxMod1 : BOOL;
	diStatusHochdruckMinMod1 : BOOL;
	diStatusHochdruckMaxMod1 : BOOL;
	diStatusNiederdruckMinMod2 : BOOL;
	diStatusNiederdruckMaxMod2 : BOOL;
	diStatusHochdruckMinMod2 : BOOL;
	diStatusHochdruckMaxMod2 : BOOL;
	diStatusDifferenzdruckMax : BOOL;
	diStatusDifferenzdruckMin : BOOL;
	diStatusLuftgeschwDrahtbruch : BOOL;
	diStatusLuftgeschwMax : BOOL;
	diStatusLuftgeschwMin : BOOL;
	diStatusEintrittTempMin : BOOL;
	diStatusEintrittTempMax : BOOL;
	diStatusEintrittFeuchteMin : BOOL;
	diStatusEintrittFeuchteMax : BOOL;
	diStatusAustrittTempMin : BOOL;
	diStatusAustrittTempMax : BOOL;
	diStatusAustrittFeuchteMin : BOOL;
	diStatusAustrittFeuchteMax : BOOL;
	diStatusFrischluftFeuchteMax : BOOL;
	diStatusFrischluftFeuchteMin : BOOL;
	diStatusFrischluftTempMax : BOOL;
	diStatusFrischluftTempMin : BOOL;
	diStatusTrockenluftFeuchteMax : BOOL;
	diStatusTrockenluftFeuchteMin : BOOL;
	diStatusTrockenluftTempMax : BOOL;
	diStatusTrockenluftTempMin : BOOL;
	diStatusDachluftFeuchteMax : BOOL;
	diStatusDachluftFeuchteMin : BOOL;
	diStatusDachluftTempMax : BOOL;
	diStatusDachluftTempMin : BOOL;
	diStatusAbluftTempMax : BOOL;
	diStatusAbluftTempMin : BOOL;
	diStatusAbluftFeuchteMax : BOOL;
	diStatusAbluftFeuchteMin : BOOL;
END_VAR
```

### InputOutput.typ
```iecst
(*============================================================================================================================================================================*)
(*================================================ STRUKTUREN IO-MODULE =====================================================================================================*)

TYPE
	modAP3131 : 	STRUCT
		PmeanT : INT;
		QmeanT : INT;
		SmeanT : INT;
		PFmeanT : INT;
		AenergyT : DINT;
		RenergyT : DINT;
		SAenergyT : UDINT;
		TrigDFT : BOOL;
		EnabEnergy : BOOL;
		ClearEnergy : BOOL;
		ForceEnergy : BOOL;
		RBClearEnergy : BOOL;
		ModulOk : BOOL;
	END_STRUCT;
	modBR7300 : 	STRUCT
		ModulOk : BOOL;
	END_STRUCT;
	modCM8281 : 	STRUCT
		di01 : BOOL;
		di02 : BOOL;
		di03 : BOOL;
		di04 : BOOL;
		do01 : BOOL;
		do02 : BOOL;
		ai01 : INT;
		ao01 : INT;
		StatusInput01 : USINT;
		ModulOk : BOOL;
	END_STRUCT;
	modAO2622 : 	STRUCT
		ao01 : INT;
		ao02 : INT;
		ModulOk : BOOL;
	END_STRUCT;
	modAI4622 : 	STRUCT
		ai01 : INT;
		ai02 : INT;
		ai03 : INT;
		ai04 : INT;
		StatusInput01 : USINT;
		ModulOk : BOOL;
	END_STRUCT;
	modAI8321 : 	STRUCT
		ai01 : INT;
		ai02 : INT;
		ai03 : INT;
		ai04 : INT;
		ai05 : INT;
		ai06 : INT;
		ai07 : INT;
		ai08 : INT;
		StatusInput01 : USINT;
		StatusInput02 : USINT;
		ModulOk : BOOL;
	END_STRUCT;
	modDO9322 : 	STRUCT
		do01 : BOOL;
		do02 : BOOL;
		do03 : BOOL;
		do04 : BOOL;
		do05 : BOOL;
		do06 : BOOL;
		do07 : BOOL;
		do08 : BOOL;
		do09 : BOOL;
		do10 : BOOL;
		do11 : BOOL;
		do12 : BOOL;
		ModulOk : BOOL;
	END_STRUCT;
	modDO8322 : 	STRUCT
		do01 : BOOL;
		do02 : BOOL;
		do03 : BOOL;
		do04 : BOOL;
		do05 : BOOL;
		do06 : BOOL;
		do07 : BOOL;
		do08 : BOOL;
		ModulOk : BOOL;
	END_STRUCT;
	modDI9371 : 	STRUCT
		di01 : BOOL;
		di02 : BOOL;
		di03 : BOOL;
		di04 : BOOL;
		di05 : BOOL;
		di06 : BOOL;
		di07 : BOOL;
		di08 : BOOL;
		di09 : BOOL;
		di10 : BOOL;
		di11 : BOOL;
		di12 : BOOL;
		ModulOk : BOOL;
	END_STRUCT;
	modDIF371 : 	STRUCT
		di01 : BOOL;
		di02 : BOOL;
		di03 : BOOL;
		di04 : BOOL;
		di05 : BOOL;
		di06 : BOOL;
		di07 : BOOL;
		di08 : BOOL;
		di09 : BOOL;
		di10 : BOOL;
		di11 : BOOL;
		di12 : BOOL;
		di13 : BOOL;
		di14 : BOOL;
		di15 : BOOL;
		di16 : BOOL;
		ModulOk : BOOL;
	END_STRUCT;
	modAT2222 : 	STRUCT
		at01 : INT;
		at02 : INT;
		StatusInput01 : USINT;
		ModulOk : BOOL;
	END_STRUCT;
END_TYPE
```

### Program Logical/IO/io304 (IEC)
